REGION Network 53: Thickness AxisZ Position Absolute Position2
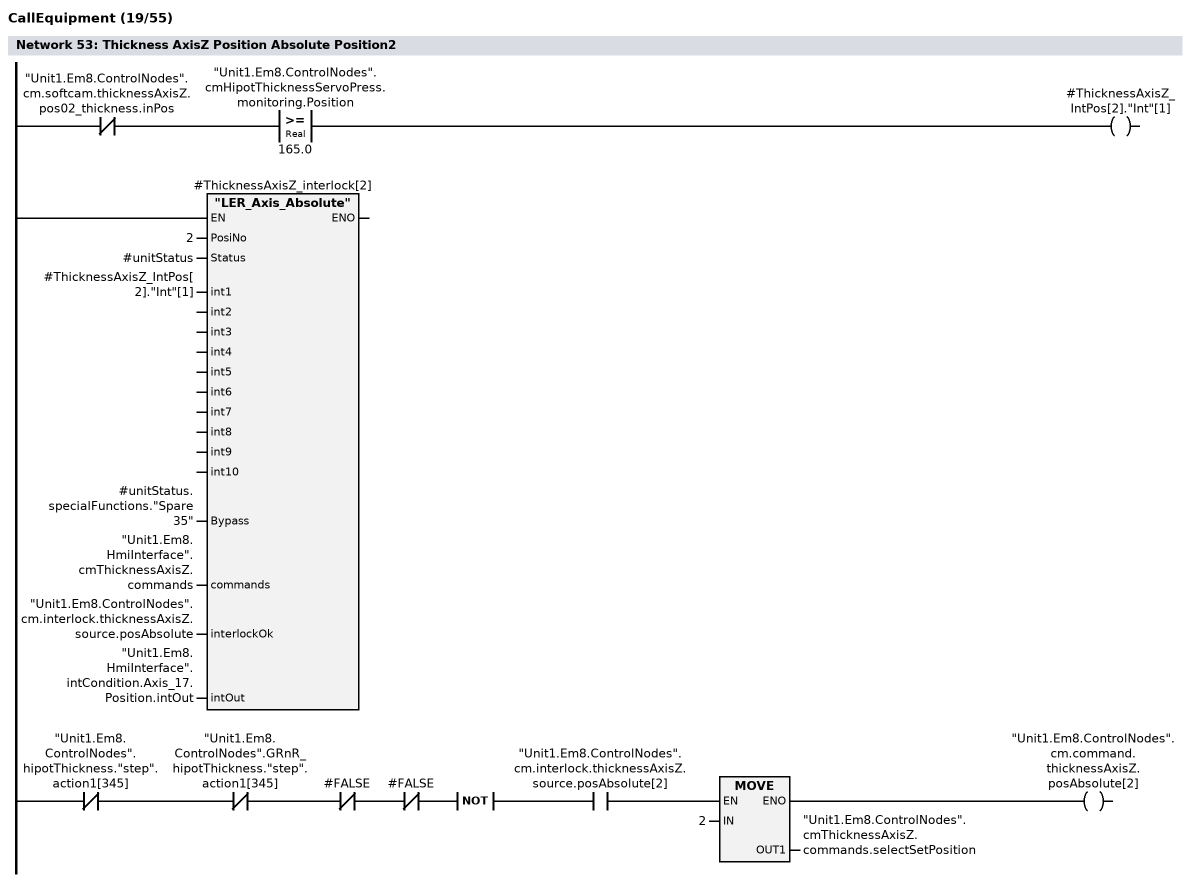
   RUNG wire#powerrail
      I_Contact( "Unit1.Em8.ControlNodes".cm.softcam.thicknessAxisZ.pos02_thickness.inPos )
      { S7_Templates := "SrcType := Real" } GE_Contact(in1 := "Unit1.Em8.ControlNodes".cmHipotThicknessServoPress.monitoring.Position, in2 := 165.0)
      Coil( #ThicknessAxisZ_IntPos[2]."Int"[1] )
   END_RUNG
   RUNG wire#powerrail
      #ThicknessAxisZ_interlock[2](PosiNo := 2, Status := #unitStatus, int1 := #ThicknessAxisZ_IntPos[2]."Int"[1], int2 :=, int3 :=, int4 :=, int5 :=, int6 :=, int7 :=, int8 :=, int9 :=, int10 :=, Bypass := #unitStatus.specialFunctions."Spare 35", commands := "Unit1.Em8.HmiInterface".cmThicknessAxisZ.commands, interlockOk := "Unit1.Em8.ControlNodes".cm.interlock.thicknessAxisZ.source.posAbsolute, intOut := "Unit1.Em8.HmiInterface".intCondition.Axis_17.Position.intOut)
   END_RUNG
   RUNG wire#powerrail
      I_Contact( "Unit1.Em8.ControlNodes".hipotThickness."step".action1[345] )
      I_Contact( "Unit1.Em8.ControlNodes".GRnR_hipotThickness."step".action1[345] )
      I_Contact( #FALSE )
      I_Contact( #FALSE )
      Not()
      Contact( "Unit1.Em8.ControlNodes".cm.interlock.thicknessAxisZ.source.posAbsolute[2] )
      Move(in := 2, out1 => "Unit1.Em8.ControlNodes".cmThicknessAxisZ.commands.selectSetPosition)
      Coil( "Unit1.Em8.ControlNodes".cm.command.thicknessAxisZ.posAbsolute[2] )
   END_RUNG
   // the same network as SCL:
   #ThicknessAxisZ_IntPos[2]."Int"[1] := NOT "Unit1.Em8.ControlNodes".cm.softcam.thicknessAxisZ.pos02_thickness.inPos AND ("Unit1.Em8.ControlNodes".cmHipotThicknessServoPress.monitoring.Position >= 165.0);
   #ThicknessAxisZ_interlock[2](PosiNo := 2,   // "LER_Axis_Absolute"
                           Status := #unitStatus,
                           int1 := #ThicknessAxisZ_IntPos[2]."Int"[1],
                           Bypass := #unitStatus.specialFunctions."Spare 35",
                           commands := "Unit1.Em8.HmiInterface".cmThicknessAxisZ.commands,
                           interlockOk := "Unit1.Em8.ControlNodes".cm.interlock.thicknessAxisZ.source.posAbsolute,
                           intOut := "Unit1.Em8.HmiInterface".intCondition.Axis_17.Position.intOut);
   #_w1 := NOT (NOT "Unit1.Em8.ControlNodes".hipotThickness."step".action1[345] AND NOT "Unit1.Em8.ControlNodes".GRnR_hipotThickness."step".action1[345] AND NOT #FALSE AND NOT #FALSE) AND "Unit1.Em8.ControlNodes".cm.interlock.thicknessAxisZ.source.posAbsolute[2];
   IF #_w1 THEN "Unit1.Em8.ControlNodes".cmThicknessAxisZ.commands.selectSetPosition := 2; END_IF;
   "Unit1.Em8.ControlNodes".cm.command.thicknessAxisZ.posAbsolute[2] := #_w1;
END_REGION

REGION Network 54: Thickness AxisZ Position Absolute Position3
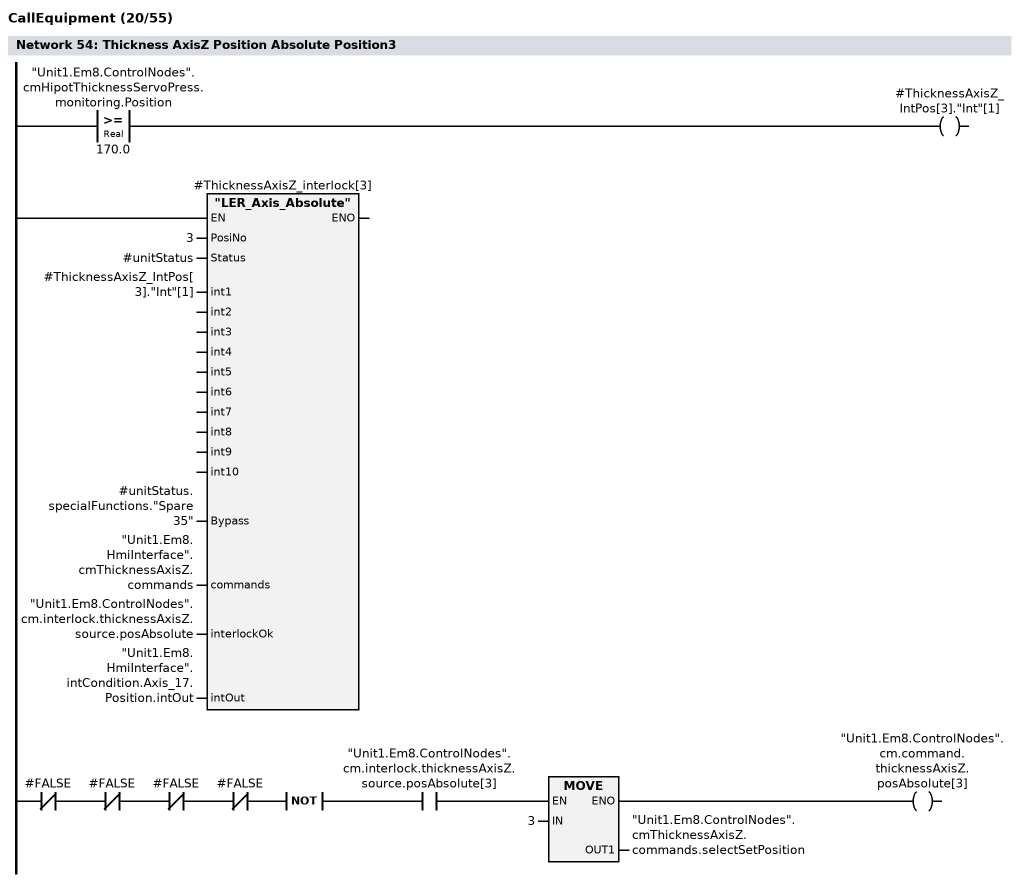
   RUNG wire#powerrail
      { S7_Templates := "SrcType := Real" } GE_Contact(in1 := "Unit1.Em8.ControlNodes".cmHipotThicknessServoPress.monitoring.Position, in2 := 170.0)
      Coil( #ThicknessAxisZ_IntPos[3]."Int"[1] )
   END_RUNG
   RUNG wire#powerrail
      #ThicknessAxisZ_interlock[3](PosiNo := 3, Status := #unitStatus, int1 := #ThicknessAxisZ_IntPos[3]."Int"[1], int2 :=, int3 :=, int4 :=, int5 :=, int6 :=, int7 :=, int8 :=, int9 :=, int10 :=, Bypass := #unitStatus.specialFunctions."Spare 35", commands := "Unit1.Em8.HmiInterface".cmThicknessAxisZ.commands, interlockOk := "Unit1.Em8.ControlNodes".cm.interlock.thicknessAxisZ.source.posAbsolute, intOut := "Unit1.Em8.HmiInterface".intCondition.Axis_17.Position.intOut)
   END_RUNG
   RUNG wire#powerrail
      I_Contact( #FALSE )
      I_Contact( #FALSE )
      I_Contact( #FALSE )
      I_Contact( #FALSE )
      Not()
      Contact( "Unit1.Em8.ControlNodes".cm.interlock.thicknessAxisZ.source.posAbsolute[3] )
      Move(in := 3, out1 => "Unit1.Em8.ControlNodes".cmThicknessAxisZ.commands.selectSetPosition)
      Coil( "Unit1.Em8.ControlNodes".cm.command.thicknessAxisZ.posAbsolute[3] )
   END_RUNG
   // the same network as SCL:
   #ThicknessAxisZ_IntPos[3]."Int"[1] := "Unit1.Em8.ControlNodes".cmHipotThicknessServoPress.monitoring.Position >= 170.0;
   #ThicknessAxisZ_interlock[3](PosiNo := 3,   // "LER_Axis_Absolute"
                           Status := #unitStatus,
                           int1 := #ThicknessAxisZ_IntPos[3]."Int"[1],
                           Bypass := #unitStatus.specialFunctions."Spare 35",
                           commands := "Unit1.Em8.HmiInterface".cmThicknessAxisZ.commands,
                           interlockOk := "Unit1.Em8.ControlNodes".cm.interlock.thicknessAxisZ.source.posAbsolute,
                           intOut := "Unit1.Em8.HmiInterface".intCondition.Axis_17.Position.intOut);
   #_w1 := NOT (NOT #FALSE AND NOT #FALSE AND NOT #FALSE AND NOT #FALSE) AND "Unit1.Em8.ControlNodes".cm.interlock.thicknessAxisZ.source.posAbsolute[3];
   IF #_w1 THEN "Unit1.Em8.ControlNodes".cmThicknessAxisZ.commands.selectSetPosition := 3; END_IF;
   "Unit1.Em8.ControlNodes".cm.command.thicknessAxisZ.posAbsolute[3] := #_w1;
END_REGION

REGION Network 55: Thickness AxisZ Position Absolute Position4
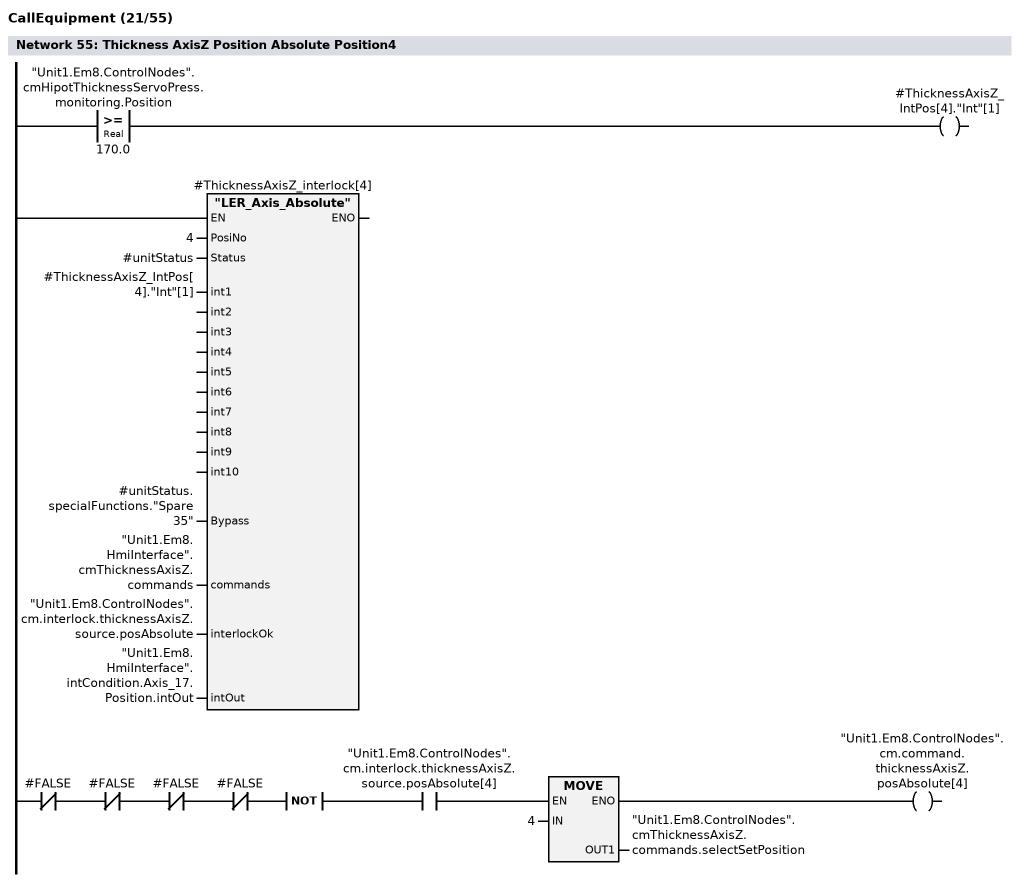
   RUNG wire#powerrail
      { S7_Templates := "SrcType := Real" } GE_Contact(in1 := "Unit1.Em8.ControlNodes".cmHipotThicknessServoPress.monitoring.Position, in2 := 170.0)
      Coil( #ThicknessAxisZ_IntPos[4]."Int"[1] )
   END_RUNG
   RUNG wire#powerrail
      #ThicknessAxisZ_interlock[4](PosiNo := 4, Status := #unitStatus, int1 := #ThicknessAxisZ_IntPos[4]."Int"[1], int2 :=, int3 :=, int4 :=, int5 :=, int6 :=, int7 :=, int8 :=, int9 :=, int10 :=, Bypass := #unitStatus.specialFunctions."Spare 35", commands := "Unit1.Em8.HmiInterface".cmThicknessAxisZ.commands, interlockOk := "Unit1.Em8.ControlNodes".cm.interlock.thicknessAxisZ.source.posAbsolute, intOut := "Unit1.Em8.HmiInterface".intCondition.Axis_17.Position.intOut)
   END_RUNG
   RUNG wire#powerrail
      I_Contact( #FALSE )
      I_Contact( #FALSE )
      I_Contact( #FALSE )
      I_Contact( #FALSE )
      Not()
      Contact( "Unit1.Em8.ControlNodes".cm.interlock.thicknessAxisZ.source.posAbsolute[4] )
      Move(in := 4, out1 => "Unit1.Em8.ControlNodes".cmThicknessAxisZ.commands.selectSetPosition)
      Coil( "Unit1.Em8.ControlNodes".cm.command.thicknessAxisZ.posAbsolute[4] )
   END_RUNG
   // the same network as SCL:
   #ThicknessAxisZ_IntPos[4]."Int"[1] := "Unit1.Em8.ControlNodes".cmHipotThicknessServoPress.monitoring.Position >= 170.0;
   #ThicknessAxisZ_interlock[4](PosiNo := 4,   // "LER_Axis_Absolute"
                           Status := #unitStatus,
                           int1 := #ThicknessAxisZ_IntPos[4]."Int"[1],
                           Bypass := #unitStatus.specialFunctions."Spare 35",
                           commands := "Unit1.Em8.HmiInterface".cmThicknessAxisZ.commands,
                           interlockOk := "Unit1.Em8.ControlNodes".cm.interlock.thicknessAxisZ.source.posAbsolute,
                           intOut := "Unit1.Em8.HmiInterface".intCondition.Axis_17.Position.intOut);
   #_w1 := NOT (NOT #FALSE AND NOT #FALSE AND NOT #FALSE AND NOT #FALSE) AND "Unit1.Em8.ControlNodes".cm.interlock.thicknessAxisZ.source.posAbsolute[4];
   IF #_w1 THEN "Unit1.Em8.ControlNodes".cmThicknessAxisZ.commands.selectSetPosition := 4; END_IF;
   "Unit1.Em8.ControlNodes".cm.command.thicknessAxisZ.posAbsolute[4] := #_w1;
END_REGION

REGION Network 56: Thickness AxisZ Position Absolute Position5
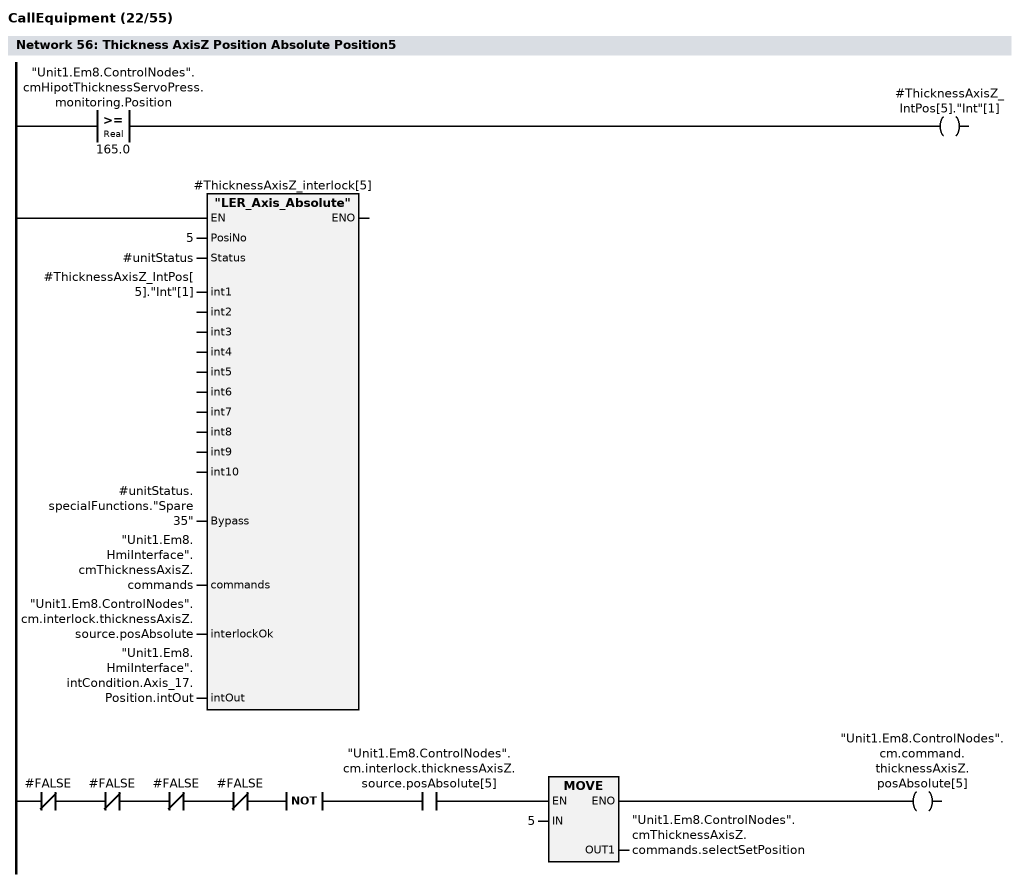
   RUNG wire#powerrail
      { S7_Templates := "SrcType := Real" } GE_Contact(in1 := "Unit1.Em8.ControlNodes".cmHipotThicknessServoPress.monitoring.Position, in2 := 165.0)
      Coil( #ThicknessAxisZ_IntPos[5]."Int"[1] )
   END_RUNG
   RUNG wire#powerrail
      #ThicknessAxisZ_interlock[5](PosiNo := 5, Status := #unitStatus, int1 := #ThicknessAxisZ_IntPos[5]."Int"[1], int2 :=, int3 :=, int4 :=, int5 :=, int6 :=, int7 :=, int8 :=, int9 :=, int10 :=, Bypass := #unitStatus.specialFunctions."Spare 35", commands := "Unit1.Em8.HmiInterface".cmThicknessAxisZ.commands, interlockOk := "Unit1.Em8.ControlNodes".cm.interlock.thicknessAxisZ.source.posAbsolute, intOut := "Unit1.Em8.HmiInterface".intCondition.Axis_17.Position.intOut)
   END_RUNG
   RUNG wire#powerrail
      I_Contact( #FALSE )
      I_Contact( #FALSE )
      I_Contact( #FALSE )
      I_Contact( #FALSE )
      Not()
      Contact( "Unit1.Em8.ControlNodes".cm.interlock.thicknessAxisZ.source.posAbsolute[5] )
      Move(in := 5, out1 => "Unit1.Em8.ControlNodes".cmThicknessAxisZ.commands.selectSetPosition)
      Coil( "Unit1.Em8.ControlNodes".cm.command.thicknessAxisZ.posAbsolute[5] )
   END_RUNG
   // the same network as SCL:
   #ThicknessAxisZ_IntPos[5]."Int"[1] := "Unit1.Em8.ControlNodes".cmHipotThicknessServoPress.monitoring.Position >= 165.0;
   #ThicknessAxisZ_interlock[5](PosiNo := 5,   // "LER_Axis_Absolute"
                           Status := #unitStatus,
                           int1 := #ThicknessAxisZ_IntPos[5]."Int"[1],
                           Bypass := #unitStatus.specialFunctions."Spare 35",
                           commands := "Unit1.Em8.HmiInterface".cmThicknessAxisZ.commands,
                           interlockOk := "Unit1.Em8.ControlNodes".cm.interlock.thicknessAxisZ.source.posAbsolute,
                           intOut := "Unit1.Em8.HmiInterface".intCondition.Axis_17.Position.intOut);
   #_w1 := NOT (NOT #FALSE AND NOT #FALSE AND NOT #FALSE AND NOT #FALSE) AND "Unit1.Em8.ControlNodes".cm.interlock.thicknessAxisZ.source.posAbsolute[5];
   IF #_w1 THEN "Unit1.Em8.ControlNodes".cmThicknessAxisZ.commands.selectSetPosition := 5; END_IF;
   "Unit1.Em8.ControlNodes".cm.command.thicknessAxisZ.posAbsolute[5] := #_w1;
END_REGION

REGION Network 57: Thickness AxisZ Position Absolute Position7
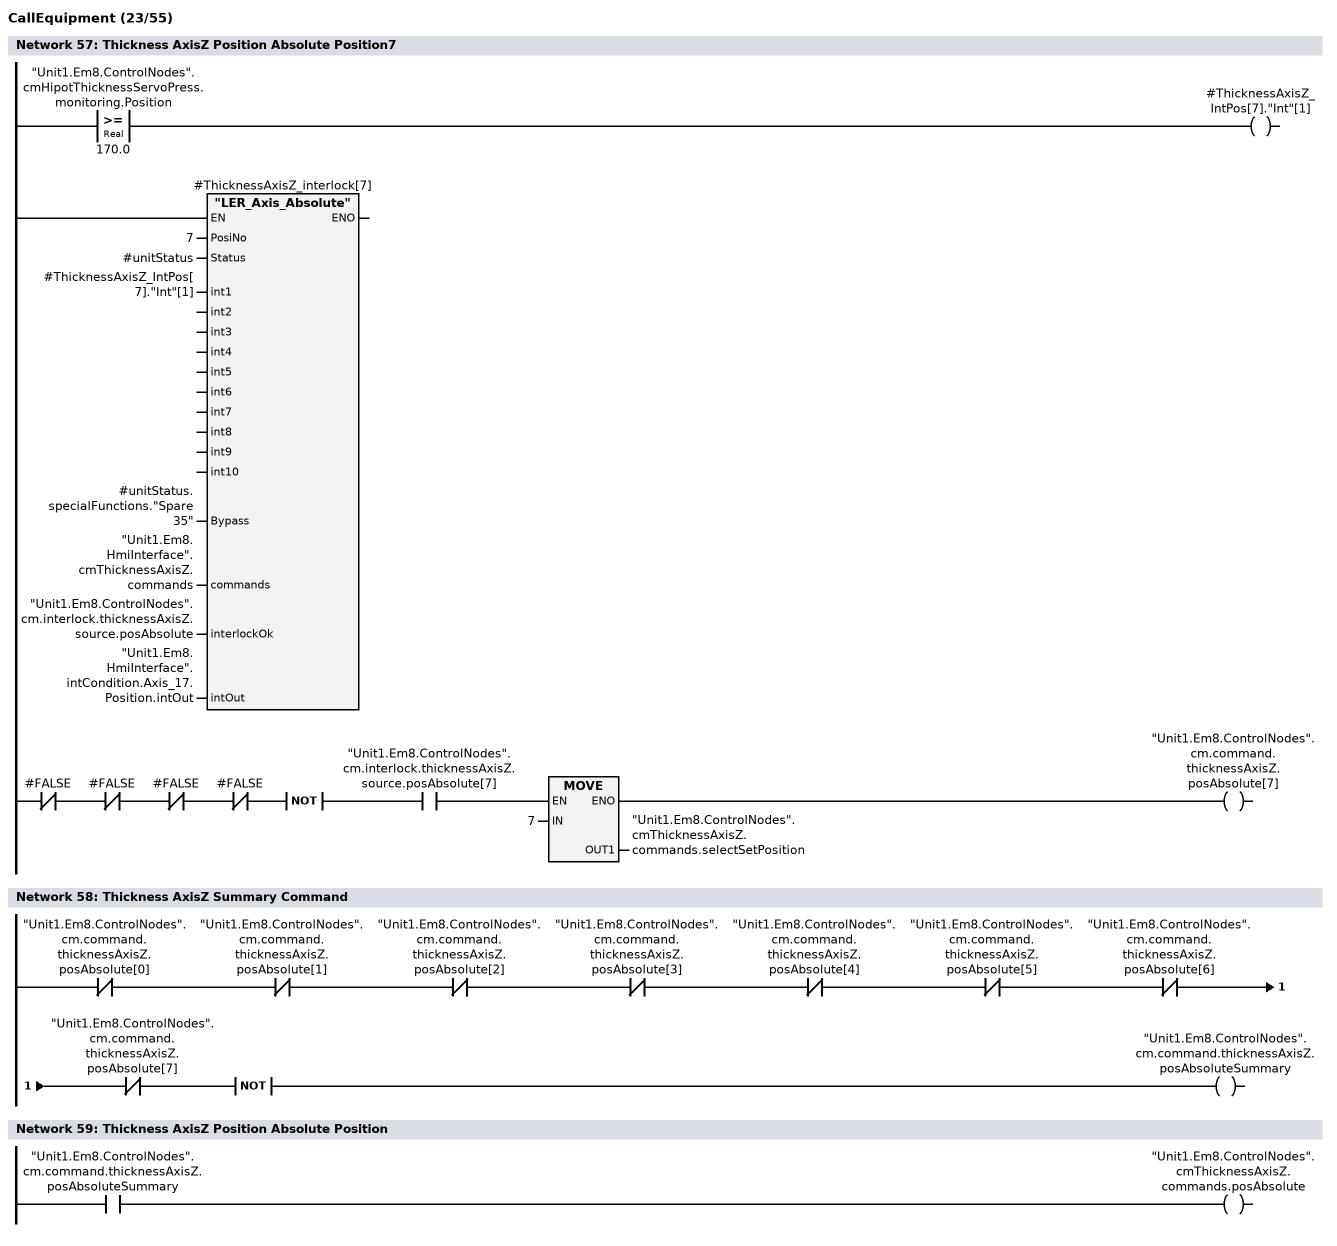
   RUNG wire#powerrail
      { S7_Templates := "SrcType := Real" } GE_Contact(in1 := "Unit1.Em8.ControlNodes".cmHipotThicknessServoPress.monitoring.Position, in2 := 170.0)
      Coil( #ThicknessAxisZ_IntPos[7]."Int"[1] )
   END_RUNG
   RUNG wire#powerrail
      #ThicknessAxisZ_interlock[7](PosiNo := 7, Status := #unitStatus, int1 := #ThicknessAxisZ_IntPos[7]."Int"[1], int2 :=, int3 :=, int4 :=, int5 :=, int6 :=, int7 :=, int8 :=, int9 :=, int10 :=, Bypass := #unitStatus.specialFunctions."Spare 35", commands := "Unit1.Em8.HmiInterface".cmThicknessAxisZ.commands, interlockOk := "Unit1.Em8.ControlNodes".cm.interlock.thicknessAxisZ.source.posAbsolute, intOut := "Unit1.Em8.HmiInterface".intCondition.Axis_17.Position.intOut)
   END_RUNG
   RUNG wire#powerrail
      I_Contact( #FALSE )
      I_Contact( #FALSE )
      I_Contact( #FALSE )
      I_Contact( #FALSE )
      Not()
      Contact( "Unit1.Em8.ControlNodes".cm.interlock.thicknessAxisZ.source.posAbsolute[7] )
      Move(in := 7, out1 => "Unit1.Em8.ControlNodes".cmThicknessAxisZ.commands.selectSetPosition)
      Coil( "Unit1.Em8.ControlNodes".cm.command.thicknessAxisZ.posAbsolute[7] )
   END_RUNG
   // the same network as SCL:
   #ThicknessAxisZ_IntPos[7]."Int"[1] := "Unit1.Em8.ControlNodes".cmHipotThicknessServoPress.monitoring.Position >= 170.0;
   #ThicknessAxisZ_interlock[7](PosiNo := 7,   // "LER_Axis_Absolute"
                           Status := #unitStatus,
                           int1 := #ThicknessAxisZ_IntPos[7]."Int"[1],
                           Bypass := #unitStatus.specialFunctions."Spare 35",
                           commands := "Unit1.Em8.HmiInterface".cmThicknessAxisZ.commands,
                           interlockOk := "Unit1.Em8.ControlNodes".cm.interlock.thicknessAxisZ.source.posAbsolute,
                           intOut := "Unit1.Em8.HmiInterface".intCondition.Axis_17.Position.intOut);
   #_w1 := NOT (NOT #FALSE AND NOT #FALSE AND NOT #FALSE AND NOT #FALSE) AND "Unit1.Em8.ControlNodes".cm.interlock.thicknessAxisZ.source.posAbsolute[7];
   IF #_w1 THEN "Unit1.Em8.ControlNodes".cmThicknessAxisZ.commands.selectSetPosition := 7; END_IF;
   "Unit1.Em8.ControlNodes".cm.command.thicknessAxisZ.posAbsolute[7] := #_w1;
END_REGION

REGION Network 58: Thickness AxisZ Summary Command
   RUNG wire#powerrail
      I_Contact( "Unit1.Em8.ControlNodes".cm.command.thicknessAxisZ.posAbsolute[0] )
      I_Contact( "Unit1.Em8.ControlNodes".cm.command.thicknessAxisZ.posAbsolute[1] )
      I_Contact( "Unit1.Em8.ControlNodes".cm.command.thicknessAxisZ.posAbsolute[2] )
      I_Contact( "Unit1.Em8.ControlNodes".cm.command.thicknessAxisZ.posAbsolute[3] )
      I_Contact( "Unit1.Em8.ControlNodes".cm.command.thicknessAxisZ.posAbsolute[4] )
      I_Contact( "Unit1.Em8.ControlNodes".cm.command.thicknessAxisZ.posAbsolute[5] )
      I_Contact( "Unit1.Em8.ControlNodes".cm.command.thicknessAxisZ.posAbsolute[6] )
      I_Contact( "Unit1.Em8.ControlNodes".cm.command.thicknessAxisZ.posAbsolute[7] )
      Not()
      Coil( "Unit1.Em8.ControlNodes".cm.command.thicknessAxisZ.posAbsoluteSummary )
   END_RUNG
   // the same network as SCL:
   "Unit1.Em8.ControlNodes".cm.command.thicknessAxisZ.posAbsoluteSummary := NOT (NOT "Unit1.Em8.ControlNodes".cm.command.thicknessAxisZ.posAbsolute[0] AND NOT "Unit1.Em8.ControlNodes".cm.command.thicknessAxisZ.posAbsolute[1] AND NOT "Unit1.Em8.ControlNodes".cm.command.thicknessAxisZ.posAbsolute[2] AND NOT "Unit1.Em8.ControlNodes".cm.command.thicknessAxisZ.posAbsolute[3] AND NOT "Unit1.Em8.ControlNodes".cm.command.thicknessAxisZ.posAbsolute[4] AND NOT "Unit1.Em8.ControlNodes".cm.command.thicknessAxisZ.posAbsolute[5] AND NOT "Unit1.Em8.ControlNodes".cm.command.thicknessAxisZ.posAbsolute[6] AND NOT "Unit1.Em8.ControlNodes".cm.command.thicknessAxisZ.posAbsolute[7]);
END_REGION

REGION Network 59: Thickness AxisZ Position Absolute Position
   RUNG wire#powerrail
      Contact( "Unit1.Em8.ControlNodes".cm.command.thicknessAxisZ.posAbsoluteSummary )
      Coil( "Unit1.Em8.ControlNodes".cmThicknessAxisZ.commands.posAbsolute )
   END_RUNG
   // the same network as SCL:
   "Unit1.Em8.ControlNodes".cmThicknessAxisZ.commands.posAbsolute := "Unit1.Em8.ControlNodes".cm.command.thicknessAxisZ.posAbsoluteSummary;
END_REGION

REGION Network 60: Thickness AxisZ Interlock Summary
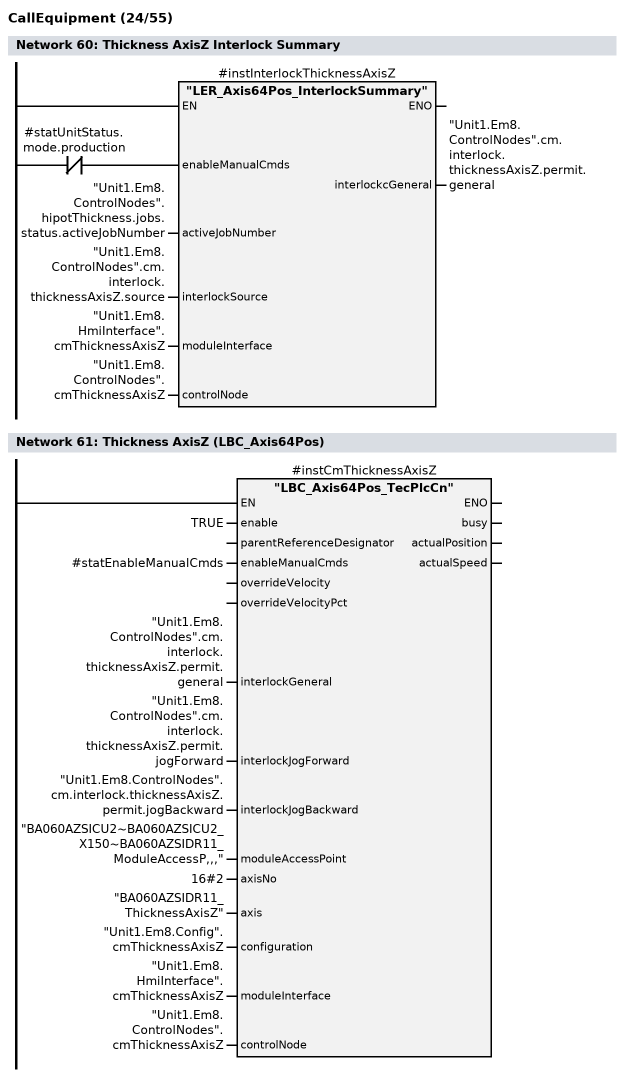
   RUNG wire#powerrail
      #instInterlockThicknessAxisZ(enableManualCmds := wire#w1, activeJobNumber := "Unit1.Em8.ControlNodes".hipotThickness.jobs.status.activeJobNumber, interlockSource := "Unit1.Em8.ControlNodes".cm.interlock.thicknessAxisZ.source, moduleInterface := "Unit1.Em8.HmiInterface".cmThicknessAxisZ, controlNode := "Unit1.Em8.ControlNodes".cmThicknessAxisZ, interlockcGeneral => "Unit1.Em8.ControlNodes".cm.interlock.thicknessAxisZ.permit.general)
   END_RUNG
   RUNG wire#powerrail
      I_Contact( #statUnitStatus.mode.production )
   END_RUNG wire#w1
   // the same network as SCL:
   #instInterlockThicknessAxisZ(enableManualCmds := NOT #statUnitStatus.mode.production,   // "LER_Axis64Pos_InterlockSummary"
                           activeJobNumber := "Unit1.Em8.ControlNodes".hipotThickness.jobs.status.activeJobNumber,
                           interlockSource := "Unit1.Em8.ControlNodes".cm.interlock.thicknessAxisZ.source,
                           moduleInterface := "Unit1.Em8.HmiInterface".cmThicknessAxisZ,
                           controlNode := "Unit1.Em8.ControlNodes".cmThicknessAxisZ,
                           interlockcGeneral => "Unit1.Em8.ControlNodes".cm.interlock.thicknessAxisZ.permit.general);
END_REGION

REGION Network 61: Thickness AxisZ (LBC_Axis64Pos)
   RUNG wire#powerrail
      #instCmThicknessAxisZ(enable := TRUE, parentReferenceDesignator :=, enableManualCmds := #statEnableManualCmds, overrideVelocity :=, overrideVelocityPct :=, interlockGeneral := "Unit1.Em8.ControlNodes".cm.interlock.thicknessAxisZ.permit.general, interlockJogForward := "Unit1.Em8.ControlNodes".cm.interlock.thicknessAxisZ.permit.jogForward, interlockJogBackward := "Unit1.Em8.ControlNodes".cm.interlock.thicknessAxisZ.permit.jogBackward, moduleAccessPoint := "BA060AZSICU2~BA060AZSICU2_X150~BA060AZSIDR11_ModuleAccessP,,,", axisNo := 16#2, axis := "BA060AZSIDR11_ThicknessAxisZ", configuration := "Unit1.Em8.Config".cmThicknessAxisZ, moduleInterface := "Unit1.Em8.HmiInterface".cmThicknessAxisZ, controlNode := "Unit1.Em8.ControlNodes".cmThicknessAxisZ, busy =>, actualPosition =>, actualSpeed =>)
   END_RUNG
   // the same network as SCL:
   #instCmThicknessAxisZ(enable := TRUE,   // "LBC_Axis64Pos_TecPlcCn"
                         enableManualCmds := #statEnableManualCmds,
                         interlockGeneral := "Unit1.Em8.ControlNodes".cm.interlock.thicknessAxisZ.permit.general,
                         interlockJogForward := "Unit1.Em8.ControlNodes".cm.interlock.thicknessAxisZ.permit.jogForward,
                         interlockJogBackward := "Unit1.Em8.ControlNodes".cm.interlock.thicknessAxisZ.permit.jogBackward,
                         moduleAccessPoint := "BA060AZSICU2~BA060AZSICU2_X150~BA060AZSIDR11_ModuleAccessP,,,",
                         axisNo := 16#2,
                         axis := "BA060AZSIDR11_ThicknessAxisZ",
                         configuration := "Unit1.Em8.Config".cmThicknessAxisZ,
                         moduleInterface := "Unit1.Em8.HmiInterface".cmThicknessAxisZ,
                         controlNode := "Unit1.Em8.ControlNodes".cmThicknessAxisZ);
END_REGION

REGION Network 62: Thickness AxisZ Softcam
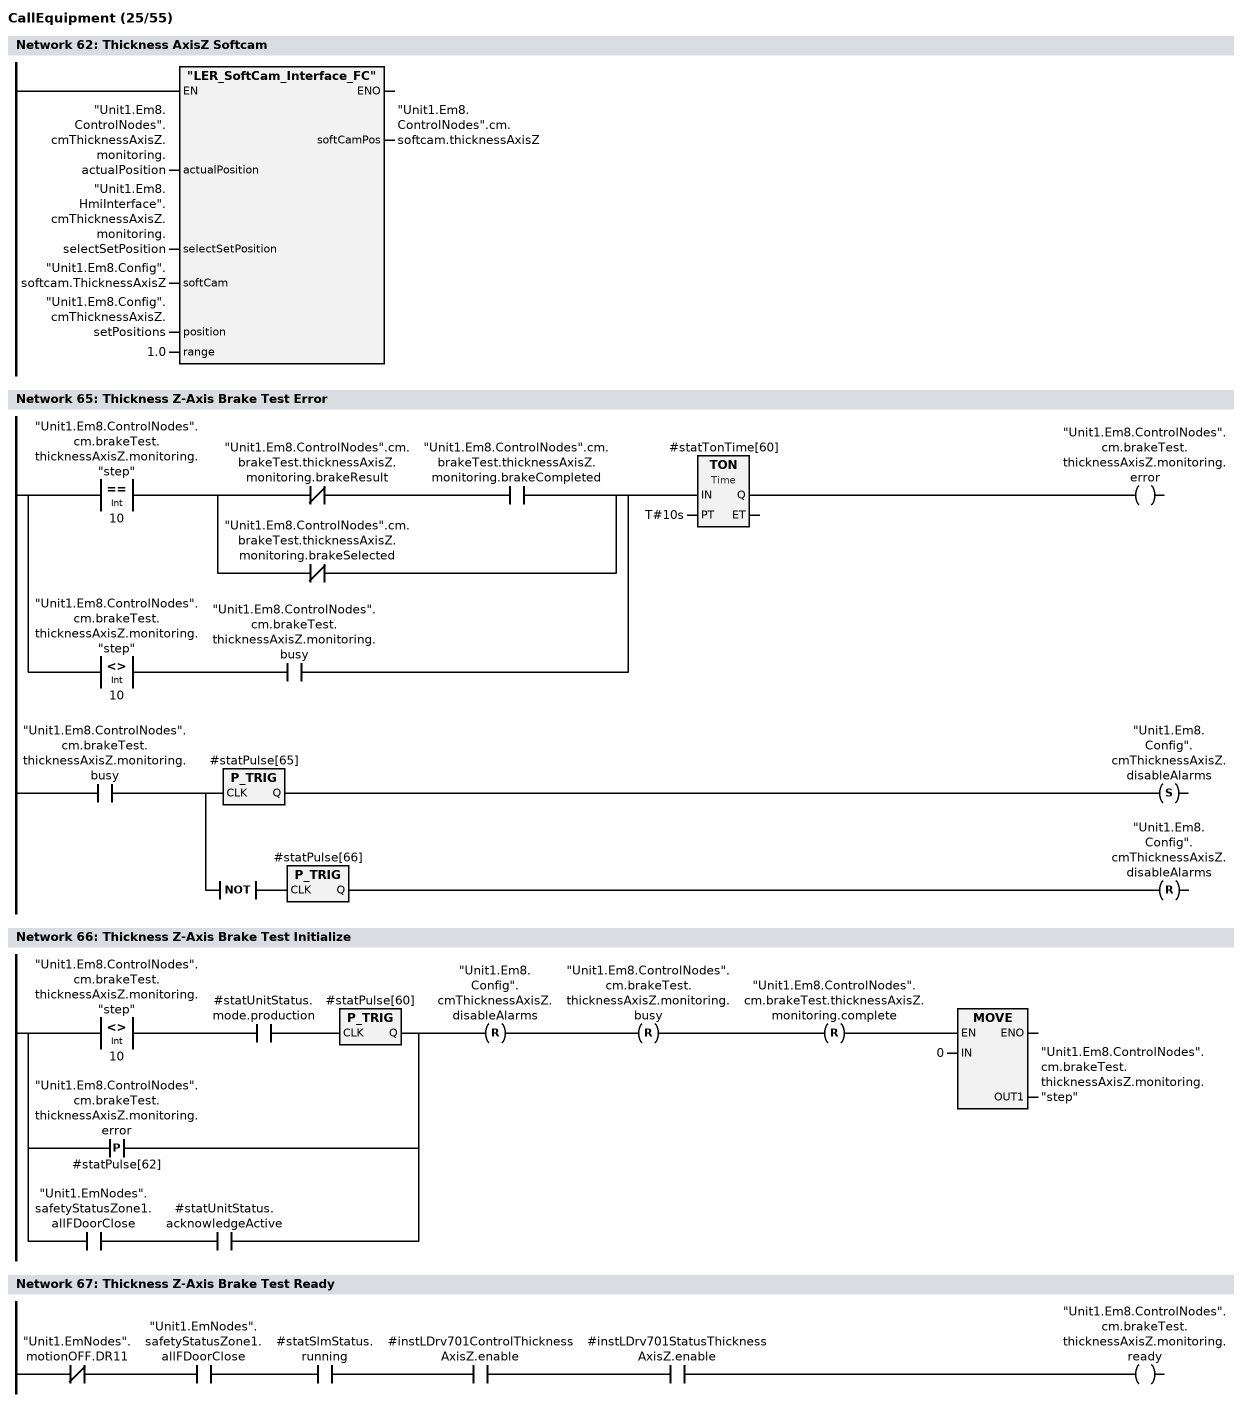
   RUNG wire#powerrail
      "LER_SoftCam_Interface_FC"(actualPosition := "Unit1.Em8.ControlNodes".cmThicknessAxisZ.monitoring.actualPosition, selectSetPosition := "Unit1.Em8.HmiInterface".cmThicknessAxisZ.monitoring.selectSetPosition, softCam := "Unit1.Em8.Config".softcam.ThicknessAxisZ, position := "Unit1.Em8.Config".cmThicknessAxisZ.setPositions, range := 1.0, softCamPos => "Unit1.Em8.ControlNodes".cm.softcam.thicknessAxisZ)
   END_RUNG
   // the same network as SCL:
   "LER_SoftCam_Interface_FC"(actualPosition := "Unit1.Em8.ControlNodes".cmThicknessAxisZ.monitoring.actualPosition,
                           selectSetPosition := "Unit1.Em8.HmiInterface".cmThicknessAxisZ.monitoring.selectSetPosition,
                           softCam := "Unit1.Em8.Config".softcam.ThicknessAxisZ,
                           position := "Unit1.Em8.Config".cmThicknessAxisZ.setPositions,
                           range := 1.0,
                           softCamPos => "Unit1.Em8.ControlNodes".cm.softcam.thicknessAxisZ);
END_REGION

REGION Network 64: ******************** Brake Test (Axis) ********************
END_REGION

REGION Network 65: Thickness Z-Axis Brake Test Error
   RUNG wire#powerrail
      { S7_Templates := "SrcType := Int" } EQ_Contact(in1 := "Unit1.Em8.ControlNodes".cm.brakeTest.thicknessAxisZ.monitoring."step", in2 := 10)
      wire#w1
      I_Contact( "Unit1.Em8.ControlNodes".cm.brakeTest.thicknessAxisZ.monitoring.brakeResult )
      Contact( "Unit1.Em8.ControlNodes".cm.brakeTest.thicknessAxisZ.monitoring.brakeCompleted )
      wire#w2
      { S7_Templates := "time_type := Time" } #statTonTime[60].TON(pt := T#10s, et =>)
      Coil( "Unit1.Em8.ControlNodes".cm.brakeTest.thicknessAxisZ.monitoring.error )
   END_RUNG
   RUNG wire#w1
      I_Contact( "Unit1.Em8.ControlNodes".cm.brakeTest.thicknessAxisZ.monitoring.brakeSelected )
   END_RUNG wire#w2
   RUNG wire#powerrail
      { S7_Templates := "SrcType := Int" } NE_Contact(in1 := "Unit1.Em8.ControlNodes".cm.brakeTest.thicknessAxisZ.monitoring."step", in2 := 10)
      Contact( "Unit1.Em8.ControlNodes".cm.brakeTest.thicknessAxisZ.monitoring.busy )
   END_RUNG wire#w2
   RUNG wire#powerrail
      Contact( "Unit1.Em8.ControlNodes".cm.brakeTest.thicknessAxisZ.monitoring.busy )
      wire#w3
      P_Trig( #statPulse[65] )
      S_Coil( "Unit1.Em8.Config".cmThicknessAxisZ.disableAlarms )
   END_RUNG
   RUNG wire#w3
      Not()
      P_Trig( #statPulse[66] )
      R_Coil( "Unit1.Em8.Config".cmThicknessAxisZ.disableAlarms )
   END_RUNG
   // the same network as SCL:
   #statTonTime[60].TON(IN := (("Unit1.Em8.ControlNodes".cm.brakeTest.thicknessAxisZ.monitoring."step" = 10) AND ((NOT "Unit1.Em8.ControlNodes".cm.brakeTest.thicknessAxisZ.monitoring.brakeResult AND "Unit1.Em8.ControlNodes".cm.brakeTest.thicknessAxisZ.monitoring.brakeCompleted) OR NOT "Unit1.Em8.ControlNodes".cm.brakeTest.thicknessAxisZ.monitoring.brakeSelected)) OR (("Unit1.Em8.ControlNodes".cm.brakeTest.thicknessAxisZ.monitoring."step" <> 10) AND "Unit1.Em8.ControlNodes".cm.brakeTest.thicknessAxisZ.monitoring.busy),
                        PT := T#10s);
   "Unit1.Em8.ControlNodes".cm.brakeTest.thicknessAxisZ.monitoring.error := #statTonTime[60].Q;
   #_w1 := "Unit1.Em8.ControlNodes".cm.brakeTest.thicknessAxisZ.monitoring.busy AND NOT #statPulse[65];   // rising edge
   #statPulse[65] := "Unit1.Em8.ControlNodes".cm.brakeTest.thicknessAxisZ.monitoring.busy;
   IF #_w1 THEN "Unit1.Em8.Config".cmThicknessAxisZ.disableAlarms := TRUE; END_IF;
   #_w2 := NOT "Unit1.Em8.ControlNodes".cm.brakeTest.thicknessAxisZ.monitoring.busy AND NOT #statPulse[66];   // rising edge
   #statPulse[66] := NOT "Unit1.Em8.ControlNodes".cm.brakeTest.thicknessAxisZ.monitoring.busy;
   IF #_w2 THEN "Unit1.Em8.Config".cmThicknessAxisZ.disableAlarms := FALSE; END_IF;
END_REGION

REGION Network 66: Thickness Z-Axis Brake Test Initialize
   RUNG wire#powerrail
      { S7_Templates := "SrcType := Int" } NE_Contact(in1 := "Unit1.Em8.ControlNodes".cm.brakeTest.thicknessAxisZ.monitoring."step", in2 := 10)
      Contact( #statUnitStatus.mode.production )
      P_Trig( #statPulse[60] )
      wire#w1
      R_Coil( "Unit1.Em8.Config".cmThicknessAxisZ.disableAlarms )
      R_Coil( "Unit1.Em8.ControlNodes".cm.brakeTest.thicknessAxisZ.monitoring.busy )
      R_Coil( "Unit1.Em8.ControlNodes".cm.brakeTest.thicknessAxisZ.monitoring.complete )
      Move(in := 0, out1 => "Unit1.Em8.ControlNodes".cm.brakeTest.thicknessAxisZ.monitoring."step")
   END_RUNG
   RUNG wire#powerrail
      P_Contact(operand := "Unit1.Em8.ControlNodes".cm.brakeTest.thicknessAxisZ.monitoring.error, bit := #statPulse[62])
   END_RUNG wire#w1
   RUNG wire#powerrail
      Contact( "Unit1.EmNodes".safetyStatusZone1.allFDoorClose )
      Contact( #statUnitStatus.acknowledgeActive )
   END_RUNG wire#w1
   // the same network as SCL:
   #_w1 := ("Unit1.Em8.ControlNodes".cm.brakeTest.thicknessAxisZ.monitoring."step" <> 10) AND #statUnitStatus.mode.production;
   #_w2 := #_w1 AND NOT #statPulse[60];   // rising edge
   #statPulse[60] := #_w1;
   #_w3 := "Unit1.Em8.ControlNodes".cm.brakeTest.thicknessAxisZ.monitoring.error AND NOT #statPulse[62];   // rising edge of "Unit1.Em8.ControlNodes".cm.brakeTest.thicknessAxisZ.monitoring.error
   #statPulse[62] := "Unit1.Em8.ControlNodes".cm.brakeTest.thicknessAxisZ.monitoring.error;
   IF #_w2 OR #_w3 OR ("Unit1.EmNodes".safetyStatusZone1.allFDoorClose AND #statUnitStatus.acknowledgeActive) THEN
       "Unit1.Em8.Config".cmThicknessAxisZ.disableAlarms := FALSE;
       "Unit1.Em8.ControlNodes".cm.brakeTest.thicknessAxisZ.monitoring.busy := FALSE;
       "Unit1.Em8.ControlNodes".cm.brakeTest.thicknessAxisZ.monitoring.complete := FALSE;
       "Unit1.Em8.ControlNodes".cm.brakeTest.thicknessAxisZ.monitoring."step" := 0;
   END_IF;
END_REGION

REGION Network 67: Thickness Z-Axis Brake Test Ready
   RUNG wire#powerrail
      I_Contact( "Unit1.EmNodes".motionOFF.DR11 )
      Contact( "Unit1.EmNodes".safetyStatusZone1.allFDoorClose )
      Contact( #statSlmStatus.running )
      Contact( #instLDrv701ControlThicknessAxisZ.enable )
      Contact( #instLDrv701StatusThicknessAxisZ.enable )
      Coil( "Unit1.Em8.ControlNodes".cm.brakeTest.thicknessAxisZ.monitoring.ready )
   END_RUNG
   // the same network as SCL:
   "Unit1.Em8.ControlNodes".cm.brakeTest.thicknessAxisZ.monitoring.ready := NOT "Unit1.EmNodes".motionOFF.DR11 AND "Unit1.EmNodes".safetyStatusZone1.allFDoorClose AND #statSlmStatus.running AND #instLDrv701ControlThicknessAxisZ.enable AND #instLDrv701StatusThicknessAxisZ.enable;
END_REGION

REGION Network 68: Thickness Z-Axis Brake Test Commands
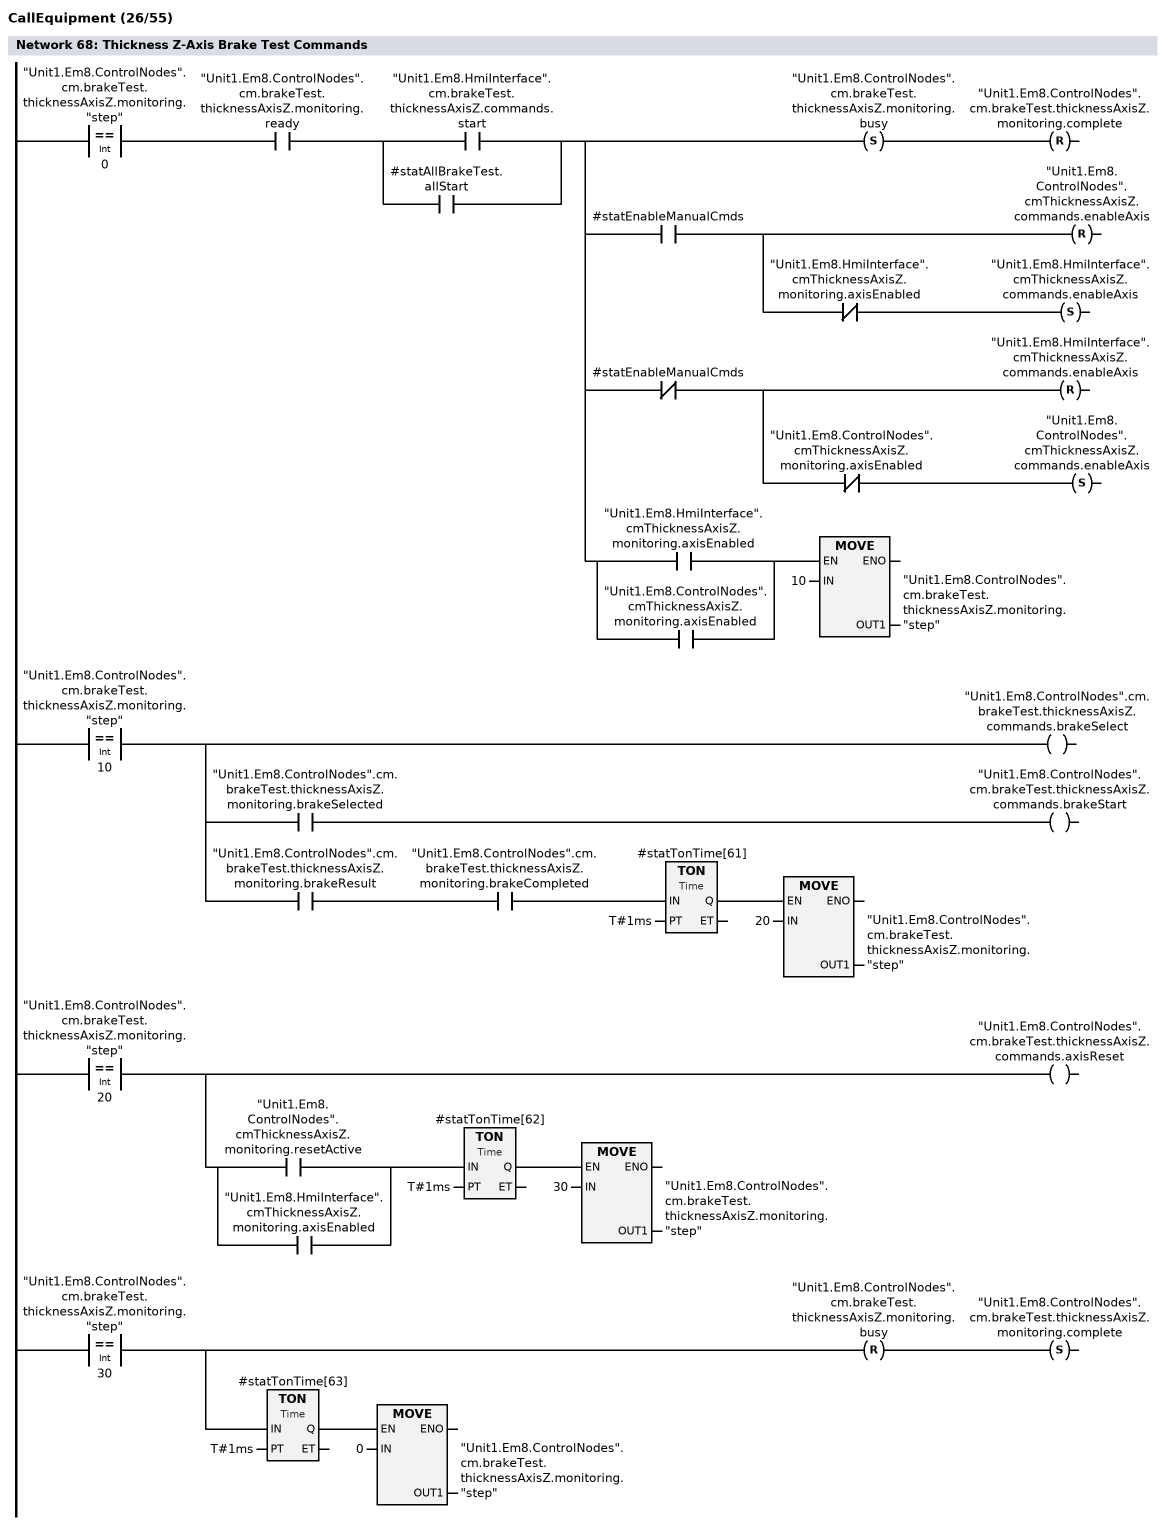
   RUNG wire#powerrail
      { S7_Templates := "SrcType := Int" } EQ_Contact(in1 := "Unit1.Em8.ControlNodes".cm.brakeTest.thicknessAxisZ.monitoring."step", in2 := 0)
      Contact( "Unit1.Em8.ControlNodes".cm.brakeTest.thicknessAxisZ.monitoring.ready )
      wire#w1
      Contact( "Unit1.Em8.HmiInterface".cm.brakeTest.thicknessAxisZ.commands.start )
      wire#w2
      S_Coil( "Unit1.Em8.ControlNodes".cm.brakeTest.thicknessAxisZ.monitoring.busy )
      R_Coil( "Unit1.Em8.ControlNodes".cm.brakeTest.thicknessAxisZ.monitoring.complete )
   END_RUNG
   RUNG wire#w1
      Contact( #statAllBrakeTest.allStart )
   END_RUNG wire#w2
   RUNG wire#w2
      Contact( #statEnableManualCmds )
      wire#w3
      R_Coil( "Unit1.Em8.ControlNodes".cmThicknessAxisZ.commands.enableAxis )
   END_RUNG
   RUNG wire#w3
      I_Contact( "Unit1.Em8.HmiInterface".cmThicknessAxisZ.monitoring.axisEnabled )
      S_Coil( "Unit1.Em8.HmiInterface".cmThicknessAxisZ.commands.enableAxis )
   END_RUNG
   RUNG wire#w2
      I_Contact( #statEnableManualCmds )
      wire#w4
      R_Coil( "Unit1.Em8.HmiInterface".cmThicknessAxisZ.commands.enableAxis )
   END_RUNG
   RUNG wire#w4
      I_Contact( "Unit1.Em8.ControlNodes".cmThicknessAxisZ.monitoring.axisEnabled )
      S_Coil( "Unit1.Em8.ControlNodes".cmThicknessAxisZ.commands.enableAxis )
   END_RUNG
   RUNG wire#w2
      Contact( "Unit1.Em8.HmiInterface".cmThicknessAxisZ.monitoring.axisEnabled )
      wire#w5
      Move(in := 10, out1 => "Unit1.Em8.ControlNodes".cm.brakeTest.thicknessAxisZ.monitoring."step")
   END_RUNG
   RUNG wire#w2
      Contact( "Unit1.Em8.ControlNodes".cmThicknessAxisZ.monitoring.axisEnabled )
   END_RUNG wire#w5
   RUNG wire#powerrail
      { S7_Templates := "SrcType := Int" } EQ_Contact(in1 := "Unit1.Em8.ControlNodes".cm.brakeTest.thicknessAxisZ.monitoring."step", in2 := 10)
      wire#w6
      Coil( "Unit1.Em8.ControlNodes".cm.brakeTest.thicknessAxisZ.commands.brakeSelect )
   END_RUNG
   RUNG wire#w6
      Contact( "Unit1.Em8.ControlNodes".cm.brakeTest.thicknessAxisZ.monitoring.brakeSelected )
      Coil( "Unit1.Em8.ControlNodes".cm.brakeTest.thicknessAxisZ.commands.brakeStart )
   END_RUNG
   RUNG wire#w6
      Contact( "Unit1.Em8.ControlNodes".cm.brakeTest.thicknessAxisZ.monitoring.brakeResult )
      Contact( "Unit1.Em8.ControlNodes".cm.brakeTest.thicknessAxisZ.monitoring.brakeCompleted )
      { S7_Templates := "time_type := Time" } #statTonTime[61].TON(pt := T#1ms, et =>)
      Move(in := 20, out1 => "Unit1.Em8.ControlNodes".cm.brakeTest.thicknessAxisZ.monitoring."step")
   END_RUNG
   RUNG wire#powerrail
      { S7_Templates := "SrcType := Int" } EQ_Contact(in1 := "Unit1.Em8.ControlNodes".cm.brakeTest.thicknessAxisZ.monitoring."step", in2 := 20)
      wire#w7
      Coil( "Unit1.Em8.ControlNodes".cm.brakeTest.thicknessAxisZ.commands.axisReset )
   END_RUNG
   RUNG wire#w7
      Contact( "Unit1.Em8.ControlNodes".cmThicknessAxisZ.monitoring.resetActive )
      wire#w8
      { S7_Templates := "time_type := Time" } #statTonTime[62].TON(pt := T#1ms, et =>)
      Move(in := 30, out1 => "Unit1.Em8.ControlNodes".cm.brakeTest.thicknessAxisZ.monitoring."step")
   END_RUNG
   RUNG wire#w7
      Contact( "Unit1.Em8.HmiInterface".cmThicknessAxisZ.monitoring.axisEnabled )
   END_RUNG wire#w8
   RUNG wire#powerrail
      { S7_Templates := "SrcType := Int" } EQ_Contact(in1 := "Unit1.Em8.ControlNodes".cm.brakeTest.thicknessAxisZ.monitoring."step", in2 := 30)
      wire#w9
      R_Coil( "Unit1.Em8.ControlNodes".cm.brakeTest.thicknessAxisZ.monitoring.busy )
      S_Coil( "Unit1.Em8.ControlNodes".cm.brakeTest.thicknessAxisZ.monitoring.complete )
   END_RUNG
   RUNG wire#w9
      { S7_Templates := "time_type := Time" } #statTonTime[63].TON(pt := T#1ms, et =>)
      Move(in := 0, out1 => "Unit1.Em8.ControlNodes".cm.brakeTest.thicknessAxisZ.monitoring."step")
   END_RUNG
   // the same network as SCL:
   #_w1 := ("Unit1.Em8.ControlNodes".cm.brakeTest.thicknessAxisZ.monitoring."step" = 0) AND "Unit1.Em8.ControlNodes".cm.brakeTest.thicknessAxisZ.monitoring.ready AND ("Unit1.Em8.HmiInterface".cm.brakeTest.thicknessAxisZ.commands.start OR #statAllBrakeTest.allStart);
   IF #_w1 THEN
       "Unit1.Em8.ControlNodes".cm.brakeTest.thicknessAxisZ.monitoring.busy := TRUE;
       "Unit1.Em8.ControlNodes".cm.brakeTest.thicknessAxisZ.monitoring.complete := FALSE;
   END_IF;
   #_w2 := #_w1 AND #statEnableManualCmds;
   IF #_w2 THEN "Unit1.Em8.ControlNodes".cmThicknessAxisZ.commands.enableAxis := FALSE; END_IF;
   IF #_w2 AND NOT "Unit1.Em8.HmiInterface".cmThicknessAxisZ.monitoring.axisEnabled THEN
       "Unit1.Em8.HmiInterface".cmThicknessAxisZ.commands.enableAxis := TRUE;
   END_IF;
   #_w3 := #_w1 AND NOT #statEnableManualCmds;
   IF #_w3 THEN "Unit1.Em8.HmiInterface".cmThicknessAxisZ.commands.enableAxis := FALSE; END_IF;
   IF #_w3 AND NOT "Unit1.Em8.ControlNodes".cmThicknessAxisZ.monitoring.axisEnabled THEN
       "Unit1.Em8.ControlNodes".cmThicknessAxisZ.commands.enableAxis := TRUE;
   END_IF;
   IF #_w1 AND ("Unit1.Em8.HmiInterface".cmThicknessAxisZ.monitoring.axisEnabled OR "Unit1.Em8.ControlNodes".cmThicknessAxisZ.monitoring.axisEnabled) THEN
       "Unit1.Em8.ControlNodes".cm.brakeTest.thicknessAxisZ.monitoring."step" := 10;
   END_IF;
   "Unit1.Em8.ControlNodes".cm.brakeTest.thicknessAxisZ.commands.brakeSelect := "Unit1.Em8.ControlNodes".cm.brakeTest.thicknessAxisZ.monitoring."step" = 10;
   "Unit1.Em8.ControlNodes".cm.brakeTest.thicknessAxisZ.commands.brakeStart := "Unit1.Em8.ControlNodes".cm.brakeTest.thicknessAxisZ.commands.brakeSelect AND "Unit1.Em8.ControlNodes".cm.brakeTest.thicknessAxisZ.monitoring.brakeSelected;
   #statTonTime[61].TON(IN := "Unit1.Em8.ControlNodes".cm.brakeTest.thicknessAxisZ.commands.brakeSelect AND "Unit1.Em8.ControlNodes".cm.brakeTest.thicknessAxisZ.monitoring.brakeResult AND "Unit1.Em8.ControlNodes".cm.brakeTest.thicknessAxisZ.monitoring.brakeCompleted,
                        PT := T#1ms);
   IF #statTonTime[61].Q THEN
       "Unit1.Em8.ControlNodes".cm.brakeTest.thicknessAxisZ.monitoring."step" := 20;
   END_IF;
   "Unit1.Em8.ControlNodes".cm.brakeTest.thicknessAxisZ.commands.axisReset := "Unit1.Em8.ControlNodes".cm.brakeTest.thicknessAxisZ.monitoring."step" = 20;
   #statTonTime[62].TON(IN := "Unit1.Em8.ControlNodes".cm.brakeTest.thicknessAxisZ.commands.axisReset AND ("Unit1.Em8.ControlNodes".cmThicknessAxisZ.monitoring.resetActive OR "Unit1.Em8.HmiInterface".cmThicknessAxisZ.monitoring.axisEnabled),
                        PT := T#1ms);
   IF #statTonTime[62].Q THEN
       "Unit1.Em8.ControlNodes".cm.brakeTest.thicknessAxisZ.monitoring."step" := 30;
   END_IF;
   #_w4 := "Unit1.Em8.ControlNodes".cm.brakeTest.thicknessAxisZ.monitoring."step" = 30;
   IF #_w4 THEN
       "Unit1.Em8.ControlNodes".cm.brakeTest.thicknessAxisZ.monitoring.busy := FALSE;
       "Unit1.Em8.ControlNodes".cm.brakeTest.thicknessAxisZ.monitoring.complete := TRUE;
   END_IF;
   #statTonTime[63].TON(IN := #_w4, PT := T#1ms);
   IF #statTonTime[63].Q THEN
       "Unit1.Em8.ControlNodes".cm.brakeTest.thicknessAxisZ.monitoring."step" := 0;
   END_IF;
END_REGION

REGION Network 69: Thickness Z-Axis Brake Test Monitoring
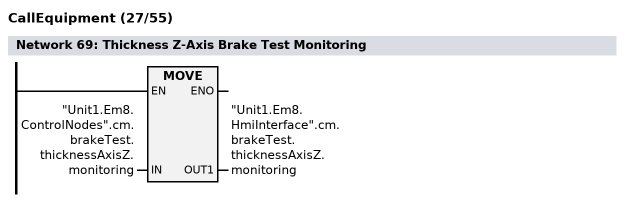
   RUNG wire#powerrail
      Move(in := "Unit1.Em8.ControlNodes".cm.brakeTest.thicknessAxisZ.monitoring, out1 => "Unit1.Em8.HmiInterface".cm.brakeTest.thicknessAxisZ.monitoring)
   END_RUNG
   // the same network as SCL:
   "Unit1.Em8.HmiInterface".cm.brakeTest.thicknessAxisZ.monitoring := "Unit1.Em8.ControlNodes".cm.brakeTest.thicknessAxisZ.monitoring;
END_REGION

REGION Network 70: Call Thickness Z-Axis Telegram 701
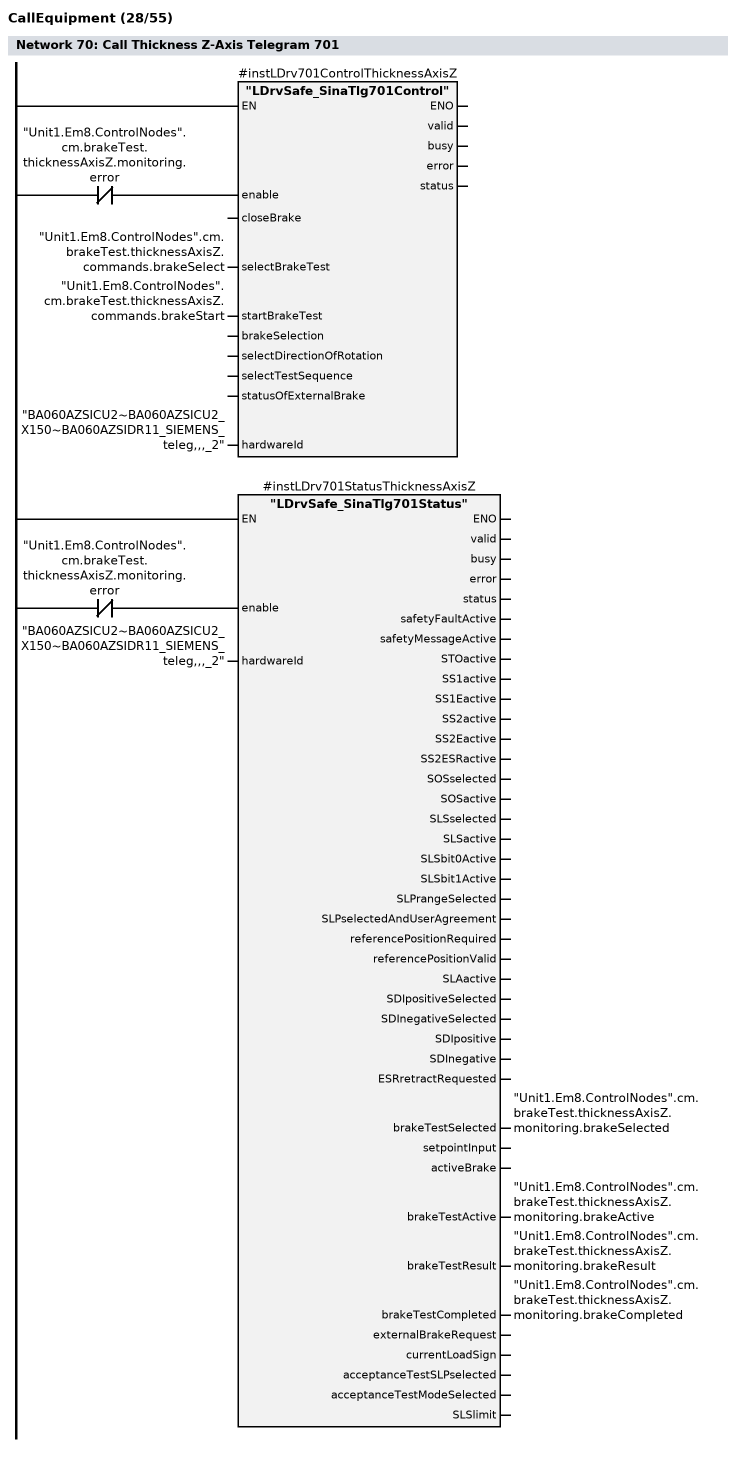
   RUNG wire#powerrail
      #instLDrv701ControlThicknessAxisZ(enable := wire#w1, closeBrake :=, selectBrakeTest := "Unit1.Em8.ControlNodes".cm.brakeTest.thicknessAxisZ.commands.brakeSelect, startBrakeTest := "Unit1.Em8.ControlNodes".cm.brakeTest.thicknessAxisZ.commands.brakeStart, brakeSelection :=, selectDirectionOfRotation :=, selectTestSequence :=, statusOfExternalBrake :=, hardwareId := "BA060AZSICU2~BA060AZSICU2_X150~BA060AZSIDR11_SIEMENS_teleg,,,_2", valid =>, busy =>, error =>, status =>)
   END_RUNG
   RUNG wire#powerrail
      I_Contact( "Unit1.Em8.ControlNodes".cm.brakeTest.thicknessAxisZ.monitoring.error )
   END_RUNG wire#w1
   RUNG wire#powerrail
      #instLDrv701StatusThicknessAxisZ(enable := wire#w2, hardwareId := "BA060AZSICU2~BA060AZSICU2_X150~BA060AZSIDR11_SIEMENS_teleg,,,_2", valid =>, busy =>, error =>, status =>, safetyFaultActive =>, safetyMessageActive =>, STOactive =>, SS1active =>, SS1Eactive =>, SS2active =>, SS2Eactive =>, SS2ESRactive =>, SOSselected =>, SOSactive =>, SLSselected =>, SLSactive =>, SLSbit0Active =>, SLSbit1Active =>, SLPrangeSelected =>, SLPselectedAndUserAgreement =>, referencePositionRequired =>, referencePositionValid =>, SLAactive =>, SDIpositiveSelected =>, SDInegativeSelected =>, SDIpositive =>, SDInegative =>, ESRretractRequested =>, brakeTestSelected => "Unit1.Em8.ControlNodes".cm.brakeTest.thicknessAxisZ.monitoring.brakeSelected, setpointInput =>, activeBrake =>, brakeTestActive => "Unit1.Em8.ControlNodes".cm.brakeTest.thicknessAxisZ.monitoring.brakeActive, brakeTestResult => "Unit1.Em8.ControlNodes".cm.brakeTest.thicknessAxisZ.monitoring.brakeResult, brakeTestCompleted => "Unit1.Em8.ControlNodes".cm.brakeTest.thicknessAxisZ.monitoring.brakeCompleted, externalBrakeRequest =>, currentLoadSign =>, acceptanceTestSLPselected =>, acceptanceTestModeSelected =>, SLSlimit =>)
   END_RUNG
   RUNG wire#powerrail
      I_Contact( "Unit1.Em8.ControlNodes".cm.brakeTest.thicknessAxisZ.monitoring.error )
   END_RUNG wire#w2
   // the same network as SCL:
   #instLDrv701ControlThicknessAxisZ(enable := NOT "Unit1.Em8.ControlNodes".cm.brakeTest.thicknessAxisZ.monitoring.error,   // "LDrvSafe_SinaTlg701Control"
                           selectBrakeTest := "Unit1.Em8.ControlNodes".cm.brakeTest.thicknessAxisZ.commands.brakeSelect,
                           startBrakeTest := "Unit1.Em8.ControlNodes".cm.brakeTest.thicknessAxisZ.commands.brakeStart,
                           hardwareId := "BA060AZSICU2~BA060AZSICU2_X150~BA060AZSIDR11_SIEMENS_teleg,,,_2");
   #instLDrv701StatusThicknessAxisZ(enable := NOT "Unit1.Em8.ControlNodes".cm.brakeTest.thicknessAxisZ.monitoring.error,   // "LDrvSafe_SinaTlg701Status"
                           hardwareId := "BA060AZSICU2~BA060AZSICU2_X150~BA060AZSIDR11_SIEMENS_teleg,,,_2",
                           brakeTestSelected => "Unit1.Em8.ControlNodes".cm.brakeTest.thicknessAxisZ.monitoring.brakeSelected,
                           brakeTestActive => "Unit1.Em8.ControlNodes".cm.brakeTest.thicknessAxisZ.monitoring.brakeActive,
                           brakeTestResult => "Unit1.Em8.ControlNodes".cm.brakeTest.thicknessAxisZ.monitoring.brakeResult,
                           brakeTestCompleted => "Unit1.Em8.ControlNodes".cm.brakeTest.thicknessAxisZ.monitoring.brakeCompleted);
END_REGION

REGION Network 72: ******************** Control Modules (TwoWayActuator) ********************
   // Call control modules that are actuators after the em logic (jobs and sequence), so that the latest commands are applied to the actuators.
END_REGION

REGION Network 73: Reset CMS
   // Reset Axis when the unit is in the resetting state.
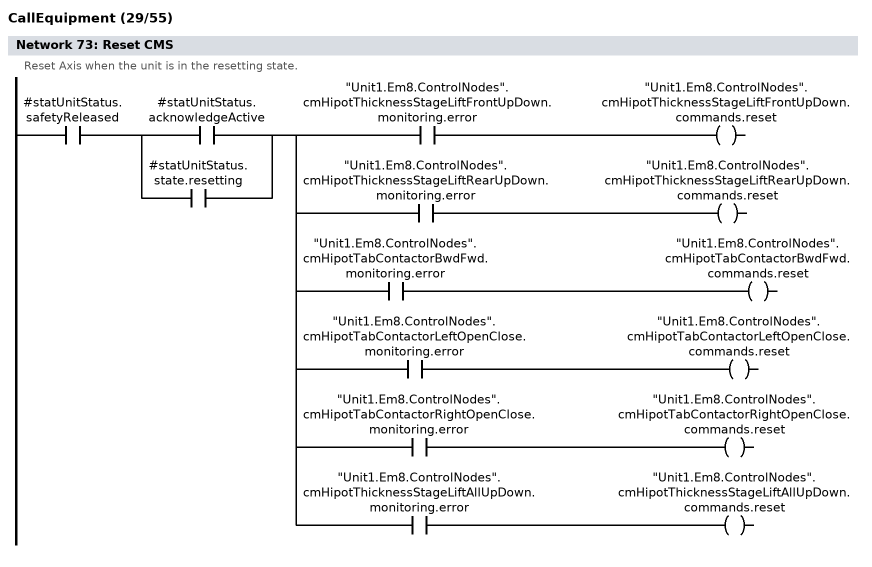
   RUNG wire#powerrail
      Contact( #statUnitStatus.safetyReleased )
      wire#w1
      Contact( #statUnitStatus.acknowledgeActive )
      wire#w2
      Contact( "Unit1.Em8.ControlNodes".cmHipotThicknessStageLiftFrontUpDown.monitoring.error )
      Coil( "Unit1.Em8.ControlNodes".cmHipotThicknessStageLiftFrontUpDown.commands.reset )
   END_RUNG
   RUNG wire#w1
      Contact( #statUnitStatus.state.resetting )
   END_RUNG wire#w2
   RUNG wire#w2
      Contact( "Unit1.Em8.ControlNodes".cmHipotThicknessStageLiftRearUpDown.monitoring.error )
      Coil( "Unit1.Em8.ControlNodes".cmHipotThicknessStageLiftRearUpDown.commands.reset )
   END_RUNG
   RUNG wire#w2
      Contact( "Unit1.Em8.ControlNodes".cmHipotTabContactorBwdFwd.monitoring.error )
      Coil( "Unit1.Em8.ControlNodes".cmHipotTabContactorBwdFwd.commands.reset )
   END_RUNG
   RUNG wire#w2
      Contact( "Unit1.Em8.ControlNodes".cmHipotTabContactorLeftOpenClose.monitoring.error )
      Coil( "Unit1.Em8.ControlNodes".cmHipotTabContactorLeftOpenClose.commands.reset )
   END_RUNG
   RUNG wire#w2
      Contact( "Unit1.Em8.ControlNodes".cmHipotTabContactorRightOpenClose.monitoring.error )
      Coil( "Unit1.Em8.ControlNodes".cmHipotTabContactorRightOpenClose.commands.reset )
   END_RUNG
   RUNG wire#w2
      Contact( "Unit1.Em8.ControlNodes".cmHipotThicknessStageLiftAllUpDown.monitoring.error )
      Coil( "Unit1.Em8.ControlNodes".cmHipotThicknessStageLiftAllUpDown.commands.reset )
   END_RUNG
   // the same network as SCL:
   #_w1 := #statUnitStatus.safetyReleased AND (#statUnitStatus.acknowledgeActive OR #statUnitStatus.state.resetting);
   "Unit1.Em8.ControlNodes".cmHipotThicknessStageLiftFrontUpDown.commands.reset := #_w1 AND "Unit1.Em8.ControlNodes".cmHipotThicknessStageLiftFrontUpDown.monitoring.error;
   "Unit1.Em8.ControlNodes".cmHipotThicknessStageLiftRearUpDown.commands.reset := #_w1 AND "Unit1.Em8.ControlNodes".cmHipotThicknessStageLiftRearUpDown.monitoring.error;
   "Unit1.Em8.ControlNodes".cmHipotTabContactorBwdFwd.commands.reset := #_w1 AND "Unit1.Em8.ControlNodes".cmHipotTabContactorBwdFwd.monitoring.error;
   "Unit1.Em8.ControlNodes".cmHipotTabContactorLeftOpenClose.commands.reset := #_w1 AND "Unit1.Em8.ControlNodes".cmHipotTabContactorLeftOpenClose.monitoring.error;
   "Unit1.Em8.ControlNodes".cmHipotTabContactorRightOpenClose.commands.reset := #_w1 AND "Unit1.Em8.ControlNodes".cmHipotTabContactorRightOpenClose.monitoring.error;
   "Unit1.Em8.ControlNodes".cmHipotThicknessStageLiftAllUpDown.commands.reset := #_w1 AND "Unit1.Em8.ControlNodes".cmHipotThicknessStageLiftAllUpDown.monitoring.error;
END_REGION

REGION Network 75: Hipot & Thickness Stage Lift Front Interlock Condition
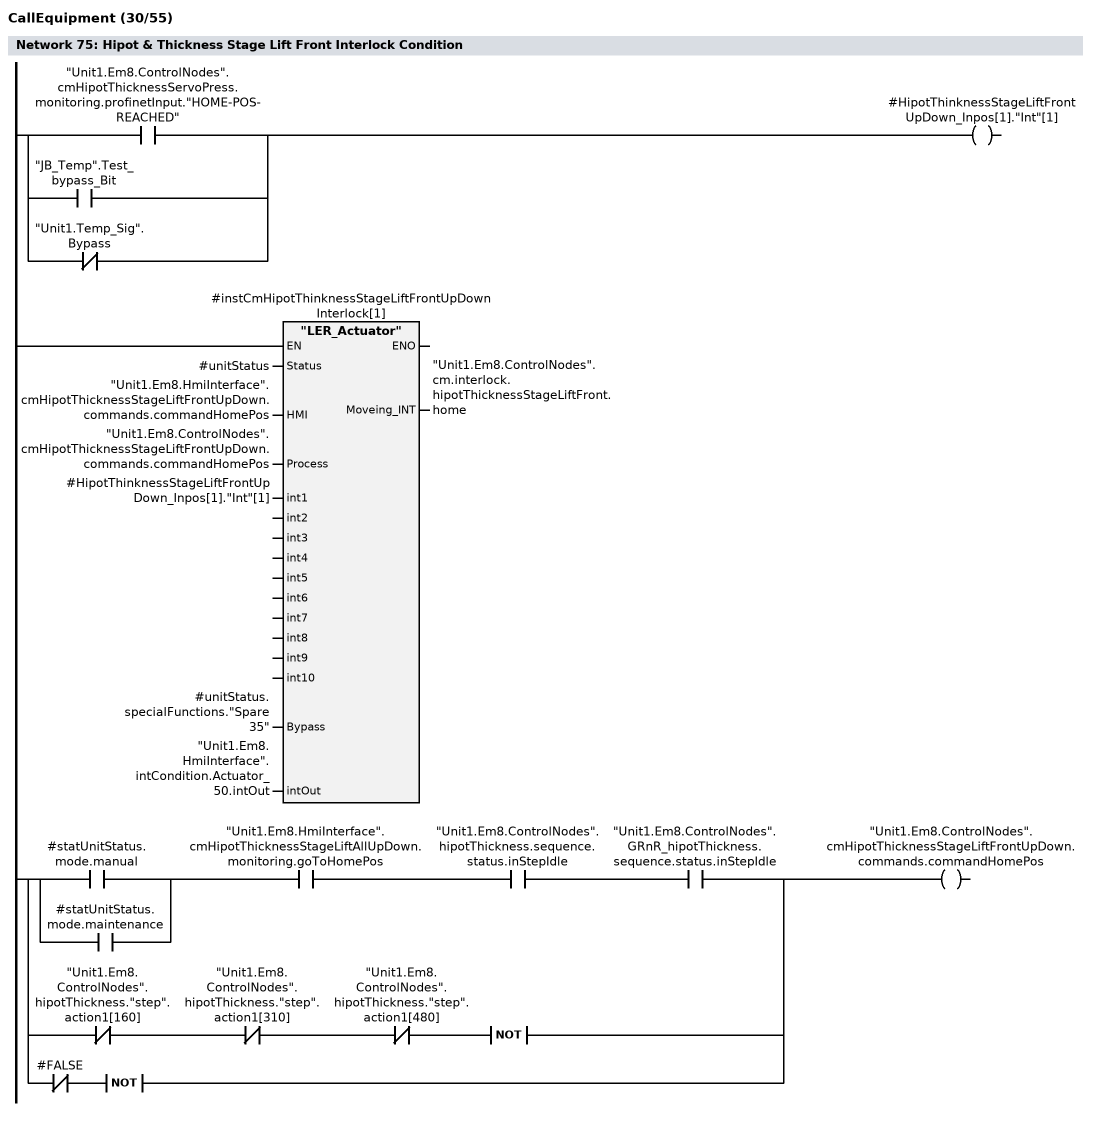
   RUNG wire#powerrail
      Contact( "Unit1.Em8.ControlNodes".cmHipotThicknessServoPress.monitoring.profinetInput."HOME-POS-REACHED" )
      wire#w1
      Coil( #HipotThinknessStageLiftFrontUpDown_Inpos[1]."Int"[1] )
   END_RUNG
   RUNG wire#powerrail
      Contact( "JB_Temp".Test_bypass_Bit )
   END_RUNG wire#w1
   RUNG wire#powerrail
      I_Contact( "Unit1.Temp_Sig".Bypass )
   END_RUNG wire#w1
   RUNG wire#powerrail
      #instCmHipotThinknessStageLiftFrontUpDownInterlock[1](Status := #unitStatus, HMI := "Unit1.Em8.HmiInterface".cmHipotThicknessStageLiftFrontUpDown.commands.commandHomePos, Process := "Unit1.Em8.ControlNodes".cmHipotThicknessStageLiftFrontUpDown.commands.commandHomePos, int1 := #HipotThinknessStageLiftFrontUpDown_Inpos[1]."Int"[1], int2 :=, int3 :=, int4 :=, int5 :=, int6 :=, int7 :=, int8 :=, int9 :=, int10 :=, Bypass := #unitStatus.specialFunctions."Spare 35", intOut := "Unit1.Em8.HmiInterface".intCondition.Actuator_50.intOut, Moveing_INT => "Unit1.Em8.ControlNodes".cm.interlock.hipotThicknessStageLiftFront.home)
   END_RUNG
   RUNG wire#powerrail
      Contact( #statUnitStatus.mode.manual )
      wire#w2
      Contact( "Unit1.Em8.HmiInterface".cmHipotThicknessStageLiftAllUpDown.monitoring.goToHomePos )
      Contact( "Unit1.Em8.ControlNodes".hipotThickness.sequence.status.inStepIdle )
      Contact( "Unit1.Em8.ControlNodes".GRnR_hipotThickness.sequence.status.inStepIdle )
      wire#w3
      Coil( "Unit1.Em8.ControlNodes".cmHipotThicknessStageLiftFrontUpDown.commands.commandHomePos )
   END_RUNG
   RUNG wire#powerrail
      Contact( #statUnitStatus.mode.maintenance )
   END_RUNG wire#w2
   RUNG wire#powerrail
      I_Contact( "Unit1.Em8.ControlNodes".hipotThickness."step".action1[160] )
      I_Contact( "Unit1.Em8.ControlNodes".hipotThickness."step".action1[310] )
      I_Contact( "Unit1.Em8.ControlNodes".hipotThickness."step".action1[480] )
      Not()
   END_RUNG wire#w3
   RUNG wire#powerrail
      I_Contact( #FALSE )
      Not()
   END_RUNG wire#w3
   // the same network as SCL:
   #HipotThinknessStageLiftFrontUpDown_Inpos[1]."Int"[1] := "Unit1.Em8.ControlNodes".cmHipotThicknessServoPress.monitoring.profinetInput."HOME-POS-REACHED" OR "JB_Temp".Test_bypass_Bit OR NOT "Unit1.Temp_Sig".Bypass;
   #instCmHipotThinknessStageLiftFrontUpDownInterlock[1](Status := #unitStatus,   // "LER_Actuator"
                           HMI := "Unit1.Em8.HmiInterface".cmHipotThicknessStageLiftFrontUpDown.commands.commandHomePos,
                           Process := "Unit1.Em8.ControlNodes".cmHipotThicknessStageLiftFrontUpDown.commands.commandHomePos,
                           int1 := #HipotThinknessStageLiftFrontUpDown_Inpos[1]."Int"[1],
                           Bypass := #unitStatus.specialFunctions."Spare 35",
                           intOut := "Unit1.Em8.HmiInterface".intCondition.Actuator_50.intOut,
                           Moveing_INT => "Unit1.Em8.ControlNodes".cm.interlock.hipotThicknessStageLiftFront.home);
   "Unit1.Em8.ControlNodes".cmHipotThicknessStageLiftFrontUpDown.commands.commandHomePos := ((#statUnitStatus.mode.manual OR #statUnitStatus.mode.maintenance) AND "Unit1.Em8.HmiInterface".cmHipotThicknessStageLiftAllUpDown.monitoring.goToHomePos AND "Unit1.Em8.ControlNodes".hipotThickness.sequence.status.inStepIdle AND "Unit1.Em8.ControlNodes".GRnR_hipotThickness.sequence.status.inStepIdle) OR NOT (NOT "Unit1.Em8.ControlNodes".hipotThickness."step".action1[160] AND NOT "Unit1.Em8.ControlNodes".hipotThickness."step".action1[310] AND NOT "Unit1.Em8.ControlNodes".hipotThickness."step".action1[480]) OR NOT (NOT #FALSE);
END_REGION

REGION Network 76: Hipot & Thickness Stage Lift Front Commands
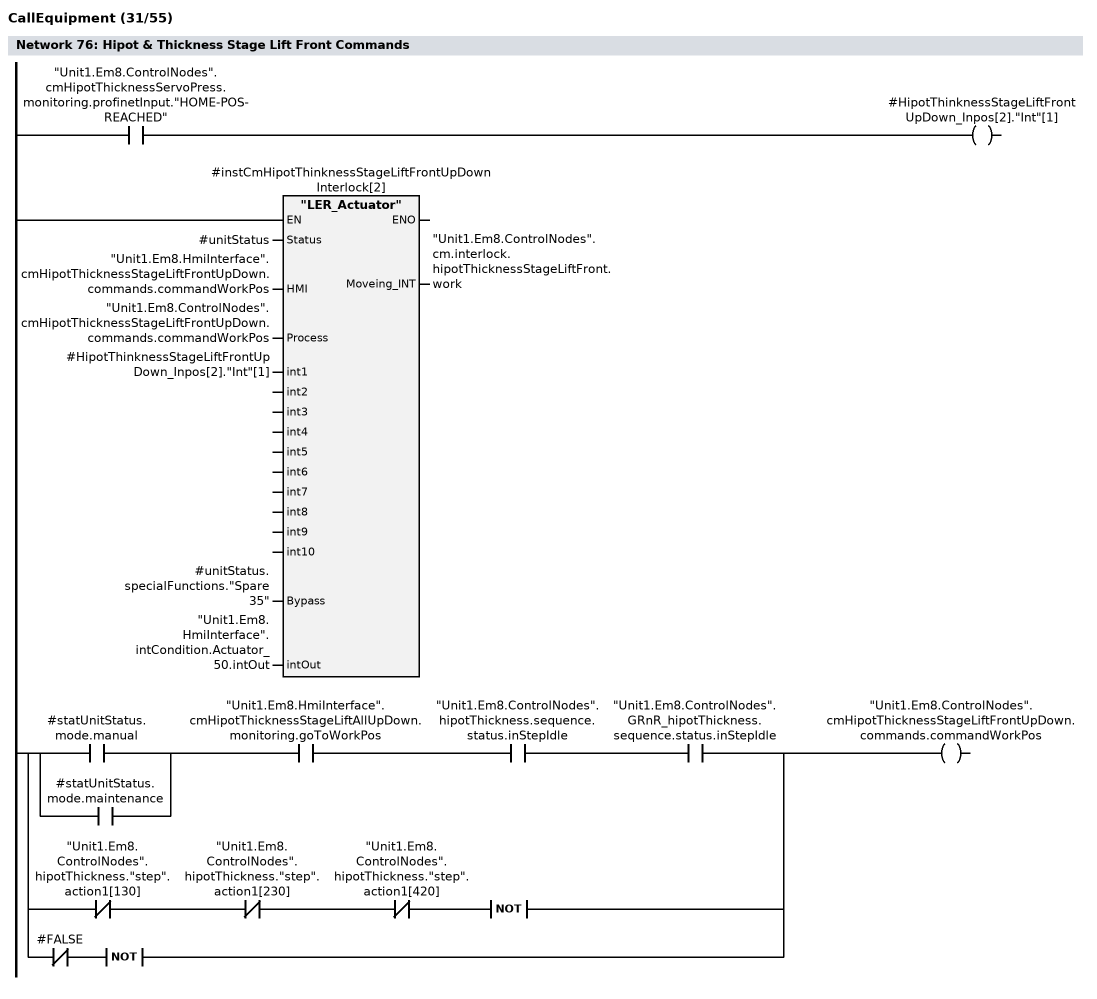
   RUNG wire#powerrail
      Contact( "Unit1.Em8.ControlNodes".cmHipotThicknessServoPress.monitoring.profinetInput."HOME-POS-REACHED" )
      Coil( #HipotThinknessStageLiftFrontUpDown_Inpos[2]."Int"[1] )
   END_RUNG
   RUNG wire#powerrail
      #instCmHipotThinknessStageLiftFrontUpDownInterlock[2](Status := #unitStatus, HMI := "Unit1.Em8.HmiInterface".cmHipotThicknessStageLiftFrontUpDown.commands.commandWorkPos, Process := "Unit1.Em8.ControlNodes".cmHipotThicknessStageLiftFrontUpDown.commands.commandWorkPos, int1 := #HipotThinknessStageLiftFrontUpDown_Inpos[2]."Int"[1], int2 :=, int3 :=, int4 :=, int5 :=, int6 :=, int7 :=, int8 :=, int9 :=, int10 :=, Bypass := #unitStatus.specialFunctions."Spare 35", intOut := "Unit1.Em8.HmiInterface".intCondition.Actuator_50.intOut, Moveing_INT => "Unit1.Em8.ControlNodes".cm.interlock.hipotThicknessStageLiftFront.work)
   END_RUNG
   RUNG wire#powerrail
      Contact( #statUnitStatus.mode.manual )
      wire#w1
      Contact( "Unit1.Em8.HmiInterface".cmHipotThicknessStageLiftAllUpDown.monitoring.goToWorkPos )
      Contact( "Unit1.Em8.ControlNodes".hipotThickness.sequence.status.inStepIdle )
      Contact( "Unit1.Em8.ControlNodes".GRnR_hipotThickness.sequence.status.inStepIdle )
      wire#w2
      Coil( "Unit1.Em8.ControlNodes".cmHipotThicknessStageLiftFrontUpDown.commands.commandWorkPos )
   END_RUNG
   RUNG wire#powerrail
      Contact( #statUnitStatus.mode.maintenance )
   END_RUNG wire#w1
   RUNG wire#powerrail
      I_Contact( "Unit1.Em8.ControlNodes".hipotThickness."step".action1[130] )
      I_Contact( "Unit1.Em8.ControlNodes".hipotThickness."step".action1[230] )
      I_Contact( "Unit1.Em8.ControlNodes".hipotThickness."step".action1[420] )
      Not()
   END_RUNG wire#w2
   RUNG wire#powerrail
      I_Contact( #FALSE )
      Not()
   END_RUNG wire#w2
   // the same network as SCL:
   #HipotThinknessStageLiftFrontUpDown_Inpos[2]."Int"[1] := "Unit1.Em8.ControlNodes".cmHipotThicknessServoPress.monitoring.profinetInput."HOME-POS-REACHED";
   #instCmHipotThinknessStageLiftFrontUpDownInterlock[2](Status := #unitStatus,   // "LER_Actuator"
                           HMI := "Unit1.Em8.HmiInterface".cmHipotThicknessStageLiftFrontUpDown.commands.commandWorkPos,
                           Process := "Unit1.Em8.ControlNodes".cmHipotThicknessStageLiftFrontUpDown.commands.commandWorkPos,
                           int1 := #HipotThinknessStageLiftFrontUpDown_Inpos[2]."Int"[1],
                           Bypass := #unitStatus.specialFunctions."Spare 35",
                           intOut := "Unit1.Em8.HmiInterface".intCondition.Actuator_50.intOut,
                           Moveing_INT => "Unit1.Em8.ControlNodes".cm.interlock.hipotThicknessStageLiftFront.work);
   "Unit1.Em8.ControlNodes".cmHipotThicknessStageLiftFrontUpDown.commands.commandWorkPos := ((#statUnitStatus.mode.manual OR #statUnitStatus.mode.maintenance) AND "Unit1.Em8.HmiInterface".cmHipotThicknessStageLiftAllUpDown.monitoring.goToWorkPos AND "Unit1.Em8.ControlNodes".hipotThickness.sequence.status.inStepIdle AND "Unit1.Em8.ControlNodes".GRnR_hipotThickness.sequence.status.inStepIdle) OR NOT (NOT "Unit1.Em8.ControlNodes".hipotThickness."step".action1[130] AND NOT "Unit1.Em8.ControlNodes".hipotThickness."step".action1[230] AND NOT "Unit1.Em8.ControlNodes".hipotThickness."step".action1[420]) OR NOT (NOT #FALSE);
END_REGION

REGION Network 77: Call CM Hipot & Thickness Stage Lift Front Cylinder Up/Down (LBC_TwoWayActuator)
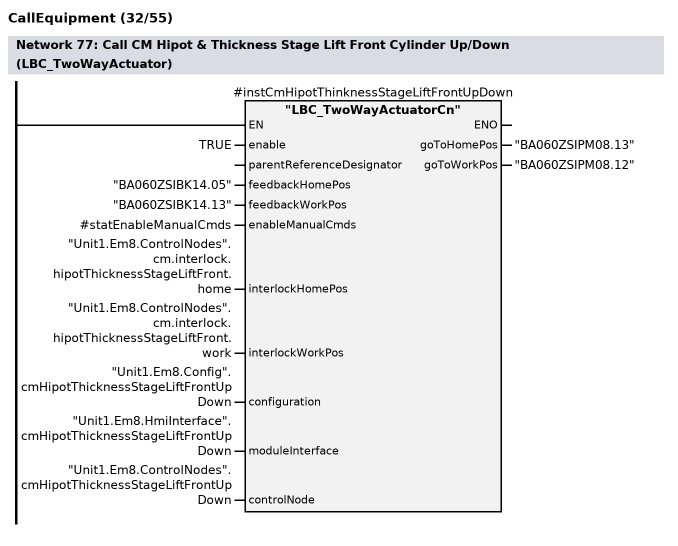
   RUNG wire#powerrail
      #instCmHipotThinknessStageLiftFrontUpDown(enable := TRUE, parentReferenceDesignator :=, feedbackHomePos := "BA060ZSIBK14.05", feedbackWorkPos := "BA060ZSIBK14.13", enableManualCmds := #statEnableManualCmds, interlockHomePos := "Unit1.Em8.ControlNodes".cm.interlock.hipotThicknessStageLiftFront.home, interlockWorkPos := "Unit1.Em8.ControlNodes".cm.interlock.hipotThicknessStageLiftFront.work, configuration := "Unit1.Em8.Config".cmHipotThicknessStageLiftFrontUpDown, moduleInterface := "Unit1.Em8.HmiInterface".cmHipotThicknessStageLiftFrontUpDown, controlNode := "Unit1.Em8.ControlNodes".cmHipotThicknessStageLiftFrontUpDown, goToHomePos => "BA060ZSIPM08.13", goToWorkPos => "BA060ZSIPM08.12")
   END_RUNG
   // the same network as SCL:
   #instCmHipotThinknessStageLiftFrontUpDown(enable := TRUE,   // "LBC_TwoWayActuatorCn"
                           feedbackHomePos := "BA060ZSIBK14.05",
                           feedbackWorkPos := "BA060ZSIBK14.13",
                           enableManualCmds := #statEnableManualCmds,
                           interlockHomePos := "Unit1.Em8.ControlNodes".cm.interlock.hipotThicknessStageLiftFront.home,
                           interlockWorkPos := "Unit1.Em8.ControlNodes".cm.interlock.hipotThicknessStageLiftFront.work,
                           configuration := "Unit1.Em8.Config".cmHipotThicknessStageLiftFrontUpDown,
                           moduleInterface := "Unit1.Em8.HmiInterface".cmHipotThicknessStageLiftFrontUpDown,
                           controlNode := "Unit1.Em8.ControlNodes".cmHipotThicknessStageLiftFrontUpDown,
                           goToHomePos => "BA060ZSIPM08.13",
                           goToWorkPos => "BA060ZSIPM08.12");
END_REGION

REGION Network 79: Hipot & Thickness Stage Lift Rear Interlock Condition
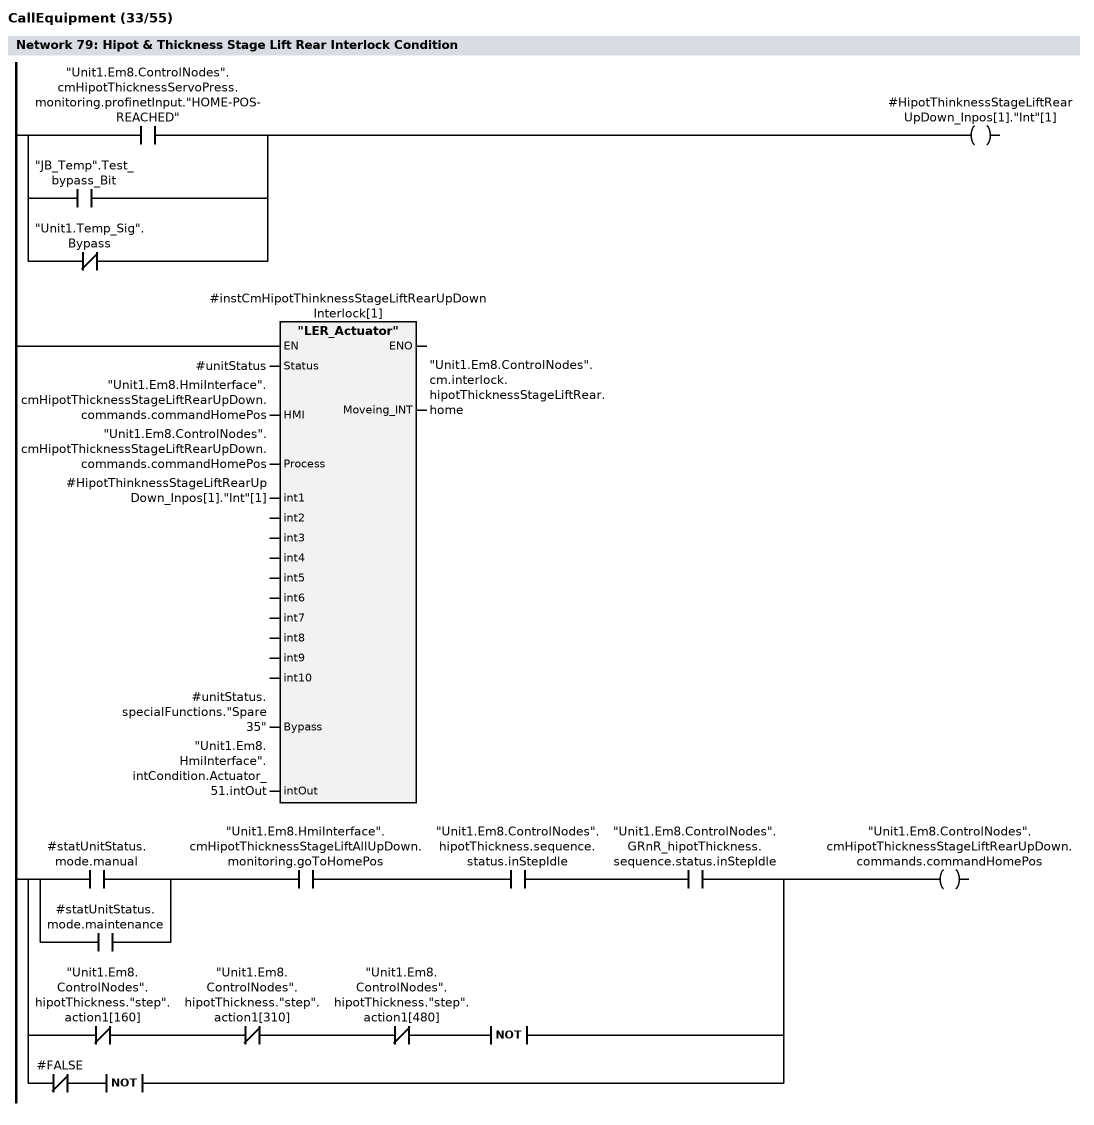
   RUNG wire#powerrail
      Contact( "Unit1.Em8.ControlNodes".cmHipotThicknessServoPress.monitoring.profinetInput."HOME-POS-REACHED" )
      wire#w1
      Coil( #HipotThinknessStageLiftRearUpDown_Inpos[1]."Int"[1] )
   END_RUNG
   RUNG wire#powerrail
      Contact( "JB_Temp".Test_bypass_Bit )
   END_RUNG wire#w1
   RUNG wire#powerrail
      I_Contact( "Unit1.Temp_Sig".Bypass )
   END_RUNG wire#w1
   RUNG wire#powerrail
      #instCmHipotThinknessStageLiftRearUpDownInterlock[1](Status := #unitStatus, HMI := "Unit1.Em8.HmiInterface".cmHipotThicknessStageLiftRearUpDown.commands.commandHomePos, Process := "Unit1.Em8.ControlNodes".cmHipotThicknessStageLiftRearUpDown.commands.commandHomePos, int1 := #HipotThinknessStageLiftRearUpDown_Inpos[1]."Int"[1], int2 :=, int3 :=, int4 :=, int5 :=, int6 :=, int7 :=, int8 :=, int9 :=, int10 :=, Bypass := #unitStatus.specialFunctions."Spare 35", intOut := "Unit1.Em8.HmiInterface".intCondition.Actuator_51.intOut, Moveing_INT => "Unit1.Em8.ControlNodes".cm.interlock.hipotThicknessStageLiftRear.home)
   END_RUNG
   RUNG wire#powerrail
      Contact( #statUnitStatus.mode.manual )
      wire#w2
      Contact( "Unit1.Em8.HmiInterface".cmHipotThicknessStageLiftAllUpDown.monitoring.goToHomePos )
      Contact( "Unit1.Em8.ControlNodes".hipotThickness.sequence.status.inStepIdle )
      Contact( "Unit1.Em8.ControlNodes".GRnR_hipotThickness.sequence.status.inStepIdle )
      wire#w3
      Coil( "Unit1.Em8.ControlNodes".cmHipotThicknessStageLiftRearUpDown.commands.commandHomePos )
   END_RUNG
   RUNG wire#powerrail
      Contact( #statUnitStatus.mode.maintenance )
   END_RUNG wire#w2
   RUNG wire#powerrail
      I_Contact( "Unit1.Em8.ControlNodes".hipotThickness."step".action1[160] )
      I_Contact( "Unit1.Em8.ControlNodes".hipotThickness."step".action1[310] )
      I_Contact( "Unit1.Em8.ControlNodes".hipotThickness."step".action1[480] )
      Not()
   END_RUNG wire#w3
   RUNG wire#powerrail
      I_Contact( #FALSE )
      Not()
   END_RUNG wire#w3
   // the same network as SCL:
   #HipotThinknessStageLiftRearUpDown_Inpos[1]."Int"[1] := "Unit1.Em8.ControlNodes".cmHipotThicknessServoPress.monitoring.profinetInput."HOME-POS-REACHED" OR "JB_Temp".Test_bypass_Bit OR NOT "Unit1.Temp_Sig".Bypass;
   #instCmHipotThinknessStageLiftRearUpDownInterlock[1](Status := #unitStatus,   // "LER_Actuator"
                           HMI := "Unit1.Em8.HmiInterface".cmHipotThicknessStageLiftRearUpDown.commands.commandHomePos,
                           Process := "Unit1.Em8.ControlNodes".cmHipotThicknessStageLiftRearUpDown.commands.commandHomePos,
                           int1 := #HipotThinknessStageLiftRearUpDown_Inpos[1]."Int"[1],
                           Bypass := #unitStatus.specialFunctions."Spare 35",
                           intOut := "Unit1.Em8.HmiInterface".intCondition.Actuator_51.intOut,
                           Moveing_INT => "Unit1.Em8.ControlNodes".cm.interlock.hipotThicknessStageLiftRear.home);
   "Unit1.Em8.ControlNodes".cmHipotThicknessStageLiftRearUpDown.commands.commandHomePos := ((#statUnitStatus.mode.manual OR #statUnitStatus.mode.maintenance) AND "Unit1.Em8.HmiInterface".cmHipotThicknessStageLiftAllUpDown.monitoring.goToHomePos AND "Unit1.Em8.ControlNodes".hipotThickness.sequence.status.inStepIdle AND "Unit1.Em8.ControlNodes".GRnR_hipotThickness.sequence.status.inStepIdle) OR NOT (NOT "Unit1.Em8.ControlNodes".hipotThickness."step".action1[160] AND NOT "Unit1.Em8.ControlNodes".hipotThickness."step".action1[310] AND NOT "Unit1.Em8.ControlNodes".hipotThickness."step".action1[480]) OR NOT (NOT #FALSE);
END_REGION

REGION Network 80: Hipot & Thickness Stage Lift Rear Commands
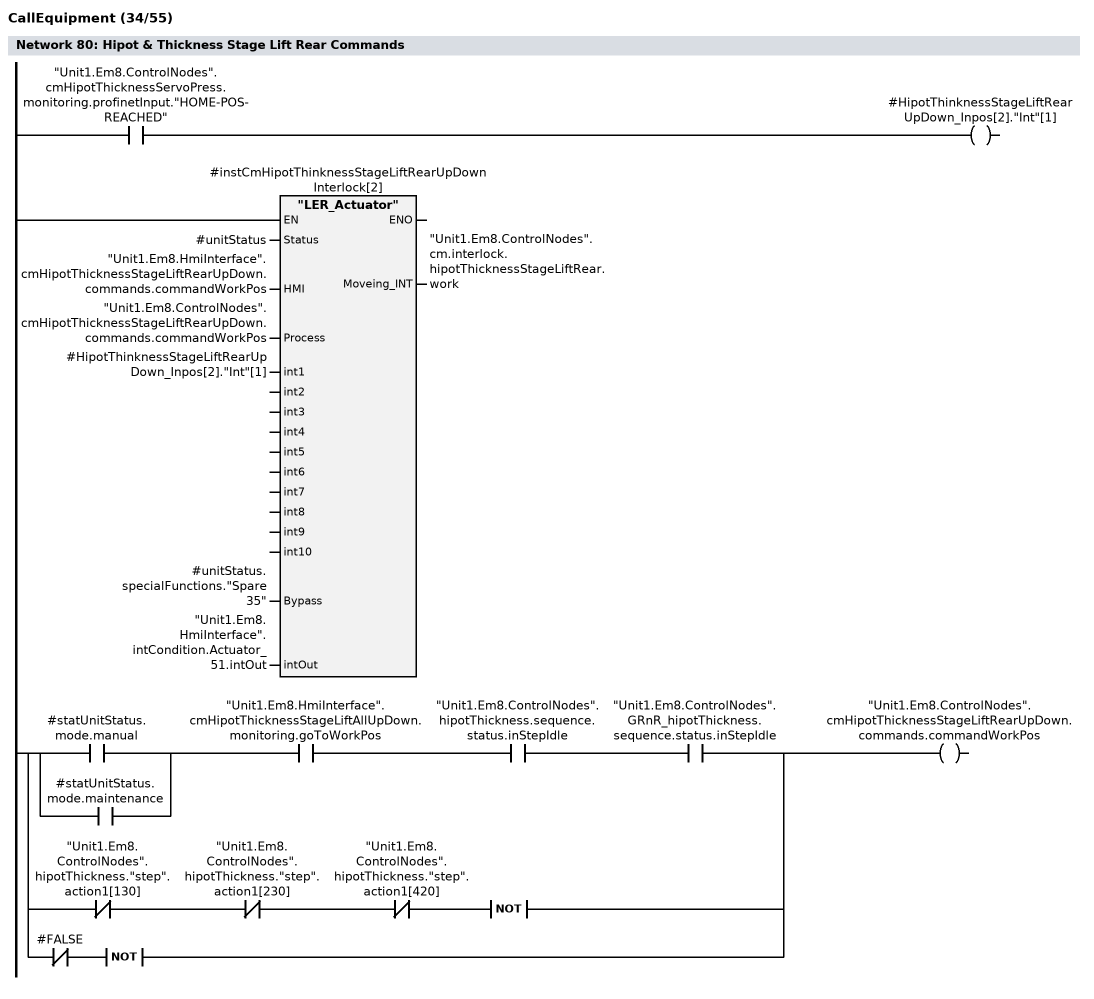
   RUNG wire#powerrail
      Contact( "Unit1.Em8.ControlNodes".cmHipotThicknessServoPress.monitoring.profinetInput."HOME-POS-REACHED" )
      Coil( #HipotThinknessStageLiftRearUpDown_Inpos[2]."Int"[1] )
   END_RUNG
   RUNG wire#powerrail
      #instCmHipotThinknessStageLiftRearUpDownInterlock[2](Status := #unitStatus, HMI := "Unit1.Em8.HmiInterface".cmHipotThicknessStageLiftRearUpDown.commands.commandWorkPos, Process := "Unit1.Em8.ControlNodes".cmHipotThicknessStageLiftRearUpDown.commands.commandWorkPos, int1 := #HipotThinknessStageLiftRearUpDown_Inpos[2]."Int"[1], int2 :=, int3 :=, int4 :=, int5 :=, int6 :=, int7 :=, int8 :=, int9 :=, int10 :=, Bypass := #unitStatus.specialFunctions."Spare 35", intOut := "Unit1.Em8.HmiInterface".intCondition.Actuator_51.intOut, Moveing_INT => "Unit1.Em8.ControlNodes".cm.interlock.hipotThicknessStageLiftRear.work)
   END_RUNG
   RUNG wire#powerrail
      Contact( #statUnitStatus.mode.manual )
      wire#w1
      Contact( "Unit1.Em8.HmiInterface".cmHipotThicknessStageLiftAllUpDown.monitoring.goToWorkPos )
      Contact( "Unit1.Em8.ControlNodes".hipotThickness.sequence.status.inStepIdle )
      Contact( "Unit1.Em8.ControlNodes".GRnR_hipotThickness.sequence.status.inStepIdle )
      wire#w2
      Coil( "Unit1.Em8.ControlNodes".cmHipotThicknessStageLiftRearUpDown.commands.commandWorkPos )
   END_RUNG
   RUNG wire#powerrail
      Contact( #statUnitStatus.mode.maintenance )
   END_RUNG wire#w1
   RUNG wire#powerrail
      I_Contact( "Unit1.Em8.ControlNodes".hipotThickness."step".action1[130] )
      I_Contact( "Unit1.Em8.ControlNodes".hipotThickness."step".action1[230] )
      I_Contact( "Unit1.Em8.ControlNodes".hipotThickness."step".action1[420] )
      Not()
   END_RUNG wire#w2
   RUNG wire#powerrail
      I_Contact( #FALSE )
      Not()
   END_RUNG wire#w2
   // the same network as SCL:
   #HipotThinknessStageLiftRearUpDown_Inpos[2]."Int"[1] := "Unit1.Em8.ControlNodes".cmHipotThicknessServoPress.monitoring.profinetInput."HOME-POS-REACHED";
   #instCmHipotThinknessStageLiftRearUpDownInterlock[2](Status := #unitStatus,   // "LER_Actuator"
                           HMI := "Unit1.Em8.HmiInterface".cmHipotThicknessStageLiftRearUpDown.commands.commandWorkPos,
                           Process := "Unit1.Em8.ControlNodes".cmHipotThicknessStageLiftRearUpDown.commands.commandWorkPos,
                           int1 := #HipotThinknessStageLiftRearUpDown_Inpos[2]."Int"[1],
                           Bypass := #unitStatus.specialFunctions."Spare 35",
                           intOut := "Unit1.Em8.HmiInterface".intCondition.Actuator_51.intOut,
                           Moveing_INT => "Unit1.Em8.ControlNodes".cm.interlock.hipotThicknessStageLiftRear.work);
   "Unit1.Em8.ControlNodes".cmHipotThicknessStageLiftRearUpDown.commands.commandWorkPos := ((#statUnitStatus.mode.manual OR #statUnitStatus.mode.maintenance) AND "Unit1.Em8.HmiInterface".cmHipotThicknessStageLiftAllUpDown.monitoring.goToWorkPos AND "Unit1.Em8.ControlNodes".hipotThickness.sequence.status.inStepIdle AND "Unit1.Em8.ControlNodes".GRnR_hipotThickness.sequence.status.inStepIdle) OR NOT (NOT "Unit1.Em8.ControlNodes".hipotThickness."step".action1[130] AND NOT "Unit1.Em8.ControlNodes".hipotThickness."step".action1[230] AND NOT "Unit1.Em8.ControlNodes".hipotThickness."step".action1[420]) OR NOT (NOT #FALSE);
END_REGION

REGION Network 81: Call CM Hipot & Thickness Stage Lift Rear Up/Down (LBC_TwoWayActuator)
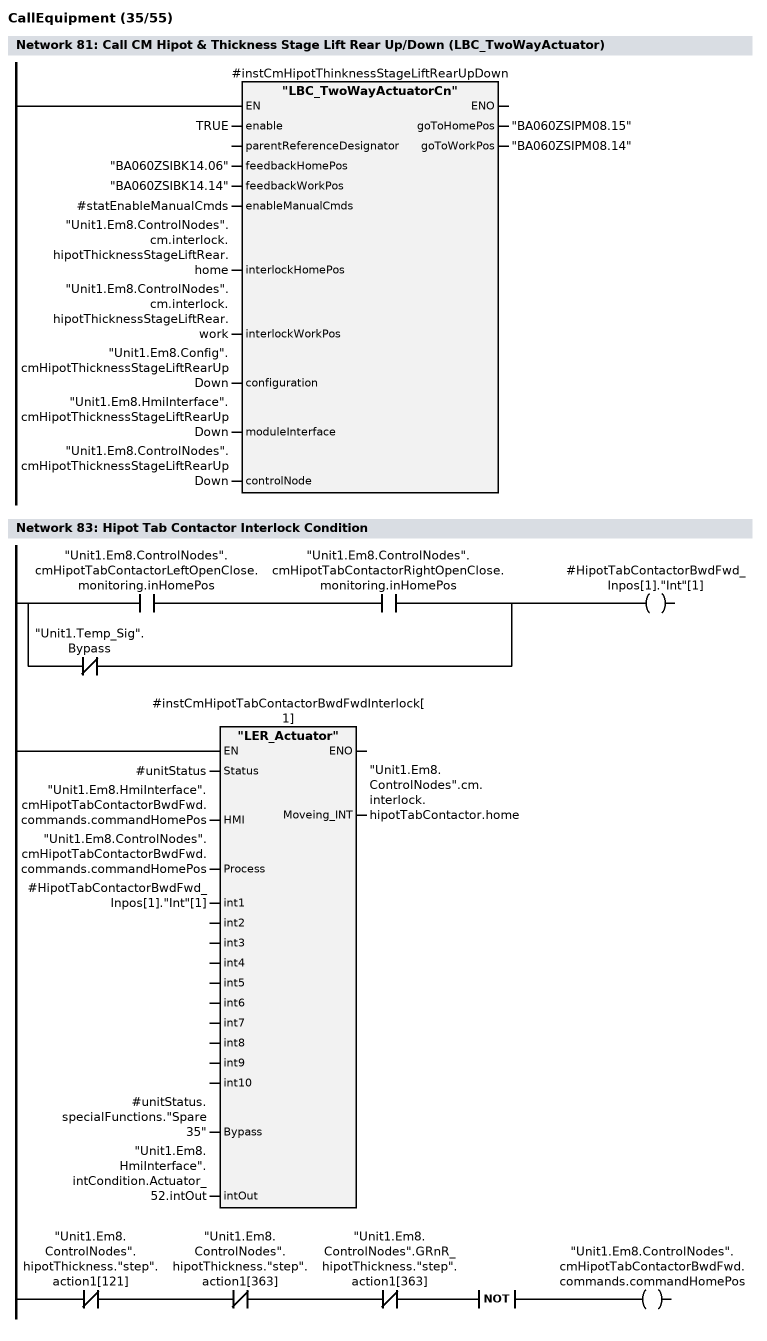
   RUNG wire#powerrail
      #instCmHipotThinknessStageLiftRearUpDown(enable := TRUE, parentReferenceDesignator :=, feedbackHomePos := "BA060ZSIBK14.06", feedbackWorkPos := "BA060ZSIBK14.14", enableManualCmds := #statEnableManualCmds, interlockHomePos := "Unit1.Em8.ControlNodes".cm.interlock.hipotThicknessStageLiftRear.home, interlockWorkPos := "Unit1.Em8.ControlNodes".cm.interlock.hipotThicknessStageLiftRear.work, configuration := "Unit1.Em8.Config".cmHipotThicknessStageLiftRearUpDown, moduleInterface := "Unit1.Em8.HmiInterface".cmHipotThicknessStageLiftRearUpDown, controlNode := "Unit1.Em8.ControlNodes".cmHipotThicknessStageLiftRearUpDown, goToHomePos => "BA060ZSIPM08.15", goToWorkPos => "BA060ZSIPM08.14")
   END_RUNG
   // the same network as SCL:
   #instCmHipotThinknessStageLiftRearUpDown(enable := TRUE,   // "LBC_TwoWayActuatorCn"
                           feedbackHomePos := "BA060ZSIBK14.06",
                           feedbackWorkPos := "BA060ZSIBK14.14",
                           enableManualCmds := #statEnableManualCmds,
                           interlockHomePos := "Unit1.Em8.ControlNodes".cm.interlock.hipotThicknessStageLiftRear.home,
                           interlockWorkPos := "Unit1.Em8.ControlNodes".cm.interlock.hipotThicknessStageLiftRear.work,
                           configuration := "Unit1.Em8.Config".cmHipotThicknessStageLiftRearUpDown,
                           moduleInterface := "Unit1.Em8.HmiInterface".cmHipotThicknessStageLiftRearUpDown,
                           controlNode := "Unit1.Em8.ControlNodes".cmHipotThicknessStageLiftRearUpDown,
                           goToHomePos => "BA060ZSIPM08.15",
                           goToWorkPos => "BA060ZSIPM08.14");
END_REGION

REGION Network 83: Hipot Tab Contactor Interlock Condition
   RUNG wire#powerrail
      Contact( "Unit1.Em8.ControlNodes".cmHipotTabContactorLeftOpenClose.monitoring.inHomePos )
      Contact( "Unit1.Em8.ControlNodes".cmHipotTabContactorRightOpenClose.monitoring.inHomePos )
      wire#w1
      Coil( #HipotTabContactorBwdFwd_Inpos[1]."Int"[1] )
   END_RUNG
   RUNG wire#powerrail
      I_Contact( "Unit1.Temp_Sig".Bypass )
   END_RUNG wire#w1
   RUNG wire#powerrail
      #instCmHipotTabContactorBwdFwdInterlock[1](Status := #unitStatus, HMI := "Unit1.Em8.HmiInterface".cmHipotTabContactorBwdFwd.commands.commandHomePos, Process := "Unit1.Em8.ControlNodes".cmHipotTabContactorBwdFwd.commands.commandHomePos, int1 := #HipotTabContactorBwdFwd_Inpos[1]."Int"[1], int2 :=, int3 :=, int4 :=, int5 :=, int6 :=, int7 :=, int8 :=, int9 :=, int10 :=, Bypass := #unitStatus.specialFunctions."Spare 35", intOut := "Unit1.Em8.HmiInterface".intCondition.Actuator_52.intOut, Moveing_INT => "Unit1.Em8.ControlNodes".cm.interlock.hipotTabContactor.home)
   END_RUNG
   RUNG wire#powerrail
      I_Contact( "Unit1.Em8.ControlNodes".hipotThickness."step".action1[121] )
      I_Contact( "Unit1.Em8.ControlNodes".hipotThickness."step".action1[363] )
      I_Contact( "Unit1.Em8.ControlNodes".GRnR_hipotThickness."step".action1[363] )
      Not()
      Coil( "Unit1.Em8.ControlNodes".cmHipotTabContactorBwdFwd.commands.commandHomePos )
   END_RUNG
   // the same network as SCL:
   #HipotTabContactorBwdFwd_Inpos[1]."Int"[1] := ("Unit1.Em8.ControlNodes".cmHipotTabContactorLeftOpenClose.monitoring.inHomePos AND "Unit1.Em8.ControlNodes".cmHipotTabContactorRightOpenClose.monitoring.inHomePos) OR NOT "Unit1.Temp_Sig".Bypass;
   #instCmHipotTabContactorBwdFwdInterlock[1](Status := #unitStatus,   // "LER_Actuator"
                           HMI := "Unit1.Em8.HmiInterface".cmHipotTabContactorBwdFwd.commands.commandHomePos,
                           Process := "Unit1.Em8.ControlNodes".cmHipotTabContactorBwdFwd.commands.commandHomePos,
                           int1 := #HipotTabContactorBwdFwd_Inpos[1]."Int"[1],
                           Bypass := #unitStatus.specialFunctions."Spare 35",
                           intOut := "Unit1.Em8.HmiInterface".intCondition.Actuator_52.intOut,
                           Moveing_INT => "Unit1.Em8.ControlNodes".cm.interlock.hipotTabContactor.home);
   "Unit1.Em8.ControlNodes".cmHipotTabContactorBwdFwd.commands.commandHomePos := NOT (NOT "Unit1.Em8.ControlNodes".hipotThickness."step".action1[121] AND NOT "Unit1.Em8.ControlNodes".hipotThickness."step".action1[363] AND NOT "Unit1.Em8.ControlNodes".GRnR_hipotThickness."step".action1[363]);
END_REGION

REGION Network 84: Hipot Tab Contactor Commands
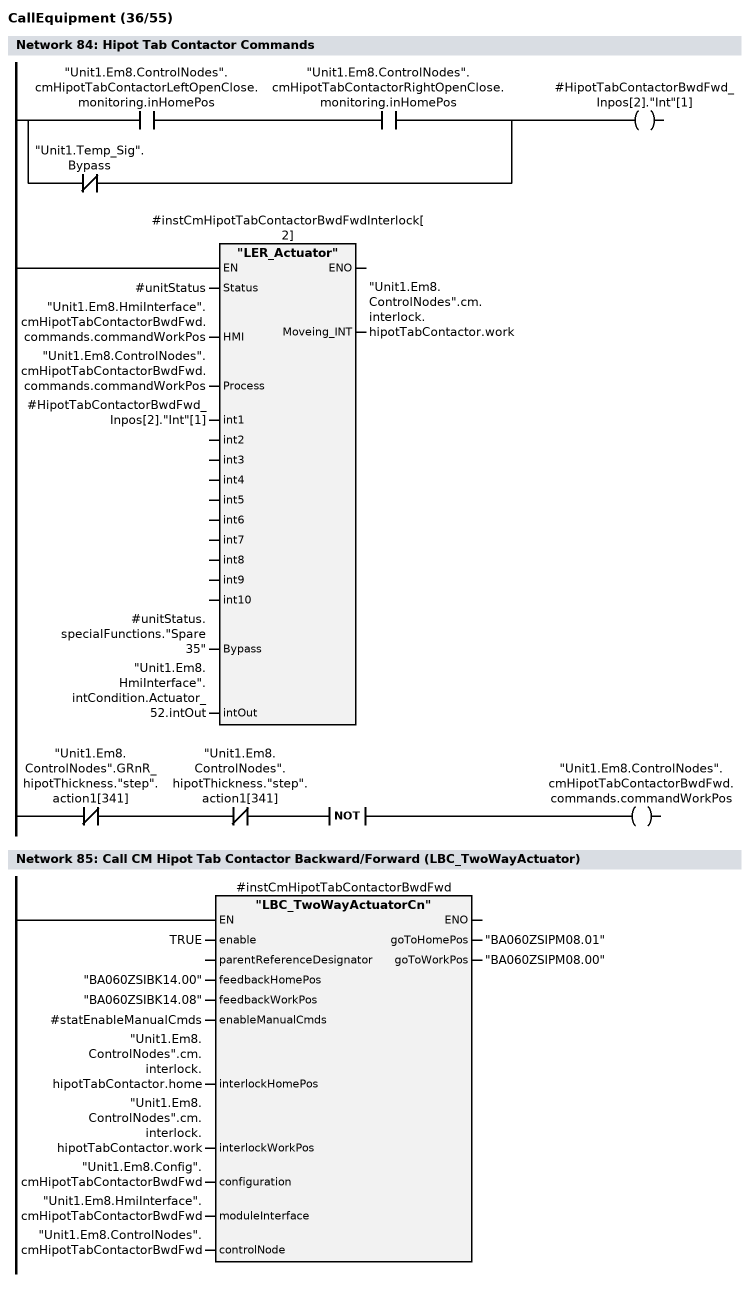
   RUNG wire#powerrail
      Contact( "Unit1.Em8.ControlNodes".cmHipotTabContactorLeftOpenClose.monitoring.inHomePos )
      Contact( "Unit1.Em8.ControlNodes".cmHipotTabContactorRightOpenClose.monitoring.inHomePos )
      wire#w1
      Coil( #HipotTabContactorBwdFwd_Inpos[2]."Int"[1] )
   END_RUNG
   RUNG wire#powerrail
      I_Contact( "Unit1.Temp_Sig".Bypass )
   END_RUNG wire#w1
   RUNG wire#powerrail
      #instCmHipotTabContactorBwdFwdInterlock[2](Status := #unitStatus, HMI := "Unit1.Em8.HmiInterface".cmHipotTabContactorBwdFwd.commands.commandWorkPos, Process := "Unit1.Em8.ControlNodes".cmHipotTabContactorBwdFwd.commands.commandWorkPos, int1 := #HipotTabContactorBwdFwd_Inpos[2]."Int"[1], int2 :=, int3 :=, int4 :=, int5 :=, int6 :=, int7 :=, int8 :=, int9 :=, int10 :=, Bypass := #unitStatus.specialFunctions."Spare 35", intOut := "Unit1.Em8.HmiInterface".intCondition.Actuator_52.intOut, Moveing_INT => "Unit1.Em8.ControlNodes".cm.interlock.hipotTabContactor.work)
   END_RUNG
   RUNG wire#powerrail
      I_Contact( "Unit1.Em8.ControlNodes".GRnR_hipotThickness."step".action1[341] )
      I_Contact( "Unit1.Em8.ControlNodes".hipotThickness."step".action1[341] )
      Not()
      Coil( "Unit1.Em8.ControlNodes".cmHipotTabContactorBwdFwd.commands.commandWorkPos )
   END_RUNG
   // the same network as SCL:
   #HipotTabContactorBwdFwd_Inpos[2]."Int"[1] := ("Unit1.Em8.ControlNodes".cmHipotTabContactorLeftOpenClose.monitoring.inHomePos AND "Unit1.Em8.ControlNodes".cmHipotTabContactorRightOpenClose.monitoring.inHomePos) OR NOT "Unit1.Temp_Sig".Bypass;
   #instCmHipotTabContactorBwdFwdInterlock[2](Status := #unitStatus,   // "LER_Actuator"
                           HMI := "Unit1.Em8.HmiInterface".cmHipotTabContactorBwdFwd.commands.commandWorkPos,
                           Process := "Unit1.Em8.ControlNodes".cmHipotTabContactorBwdFwd.commands.commandWorkPos,
                           int1 := #HipotTabContactorBwdFwd_Inpos[2]."Int"[1],
                           Bypass := #unitStatus.specialFunctions."Spare 35",
                           intOut := "Unit1.Em8.HmiInterface".intCondition.Actuator_52.intOut,
                           Moveing_INT => "Unit1.Em8.ControlNodes".cm.interlock.hipotTabContactor.work);
   "Unit1.Em8.ControlNodes".cmHipotTabContactorBwdFwd.commands.commandWorkPos := NOT (NOT "Unit1.Em8.ControlNodes".GRnR_hipotThickness."step".action1[341] AND NOT "Unit1.Em8.ControlNodes".hipotThickness."step".action1[341]);
END_REGION

REGION Network 85: Call CM Hipot Tab Contactor Backward/Forward (LBC_TwoWayActuator)
   RUNG wire#powerrail
      #instCmHipotTabContactorBwdFwd(enable := TRUE, parentReferenceDesignator :=, feedbackHomePos := "BA060ZSIBK14.00", feedbackWorkPos := "BA060ZSIBK14.08", enableManualCmds := #statEnableManualCmds, interlockHomePos := "Unit1.Em8.ControlNodes".cm.interlock.hipotTabContactor.home, interlockWorkPos := "Unit1.Em8.ControlNodes".cm.interlock.hipotTabContactor.work, configuration := "Unit1.Em8.Config".cmHipotTabContactorBwdFwd, moduleInterface := "Unit1.Em8.HmiInterface".cmHipotTabContactorBwdFwd, controlNode := "Unit1.Em8.ControlNodes".cmHipotTabContactorBwdFwd, goToHomePos => "BA060ZSIPM08.01", goToWorkPos => "BA060ZSIPM08.00")
   END_RUNG
   // the same network as SCL:
   #instCmHipotTabContactorBwdFwd(enable := TRUE,   // "LBC_TwoWayActuatorCn"
                           feedbackHomePos := "BA060ZSIBK14.00",
                           feedbackWorkPos := "BA060ZSIBK14.08",
                           enableManualCmds := #statEnableManualCmds,
                           interlockHomePos := "Unit1.Em8.ControlNodes".cm.interlock.hipotTabContactor.home,
                           interlockWorkPos := "Unit1.Em8.ControlNodes".cm.interlock.hipotTabContactor.work,
                           configuration := "Unit1.Em8.Config".cmHipotTabContactorBwdFwd,
                           moduleInterface := "Unit1.Em8.HmiInterface".cmHipotTabContactorBwdFwd,
                           controlNode := "Unit1.Em8.ControlNodes".cmHipotTabContactorBwdFwd,
                           goToHomePos => "BA060ZSIPM08.01",
                           goToWorkPos => "BA060ZSIPM08.00");
END_REGION

REGION Network 87: Hipot Tab Contactor Left Interlock Condition
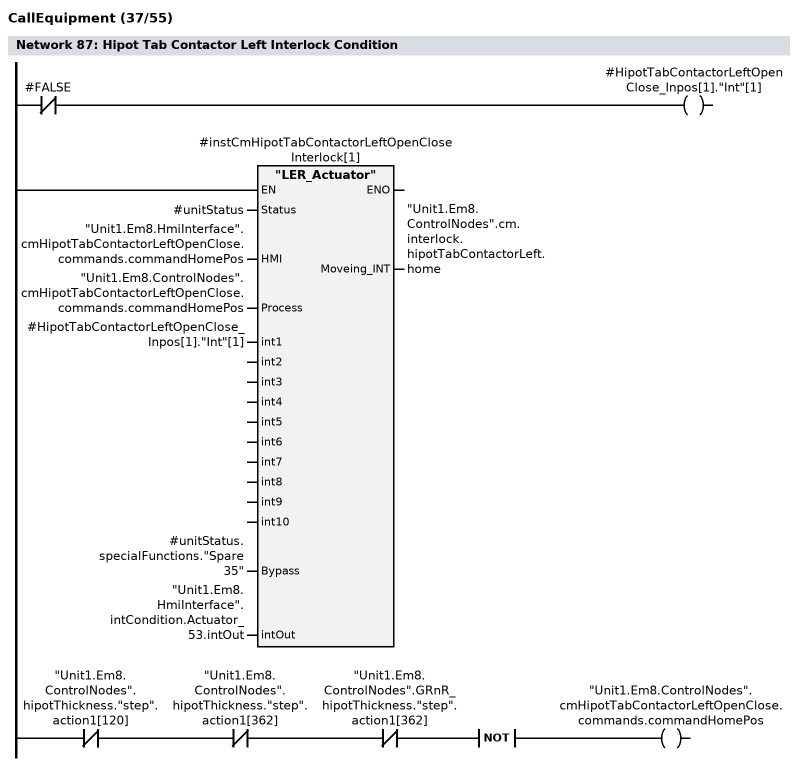
   RUNG wire#powerrail
      I_Contact( #FALSE )
      Coil( #HipotTabContactorLeftOpenClose_Inpos[1]."Int"[1] )
   END_RUNG
   RUNG wire#powerrail
      #instCmHipotTabContactorLeftOpenCloseInterlock[1](Status := #unitStatus, HMI := "Unit1.Em8.HmiInterface".cmHipotTabContactorLeftOpenClose.commands.commandHomePos, Process := "Unit1.Em8.ControlNodes".cmHipotTabContactorLeftOpenClose.commands.commandHomePos, int1 := #HipotTabContactorLeftOpenClose_Inpos[1]."Int"[1], int2 :=, int3 :=, int4 :=, int5 :=, int6 :=, int7 :=, int8 :=, int9 :=, int10 :=, Bypass := #unitStatus.specialFunctions."Spare 35", intOut := "Unit1.Em8.HmiInterface".intCondition.Actuator_53.intOut, Moveing_INT => "Unit1.Em8.ControlNodes".cm.interlock.hipotTabContactorLeft.home)
   END_RUNG
   RUNG wire#powerrail
      I_Contact( "Unit1.Em8.ControlNodes".hipotThickness."step".action1[120] )
      I_Contact( "Unit1.Em8.ControlNodes".hipotThickness."step".action1[362] )
      I_Contact( "Unit1.Em8.ControlNodes".GRnR_hipotThickness."step".action1[362] )
      Not()
      Coil( "Unit1.Em8.ControlNodes".cmHipotTabContactorLeftOpenClose.commands.commandHomePos )
   END_RUNG
   // the same network as SCL:
   #HipotTabContactorLeftOpenClose_Inpos[1]."Int"[1] := NOT #FALSE;
   #instCmHipotTabContactorLeftOpenCloseInterlock[1](Status := #unitStatus,   // "LER_Actuator"
                           HMI := "Unit1.Em8.HmiInterface".cmHipotTabContactorLeftOpenClose.commands.commandHomePos,
                           Process := "Unit1.Em8.ControlNodes".cmHipotTabContactorLeftOpenClose.commands.commandHomePos,
                           int1 := #HipotTabContactorLeftOpenClose_Inpos[1]."Int"[1],
                           Bypass := #unitStatus.specialFunctions."Spare 35",
                           intOut := "Unit1.Em8.HmiInterface".intCondition.Actuator_53.intOut,
                           Moveing_INT => "Unit1.Em8.ControlNodes".cm.interlock.hipotTabContactorLeft.home);
   "Unit1.Em8.ControlNodes".cmHipotTabContactorLeftOpenClose.commands.commandHomePos := NOT (NOT "Unit1.Em8.ControlNodes".hipotThickness."step".action1[120] AND NOT "Unit1.Em8.ControlNodes".hipotThickness."step".action1[362] AND NOT "Unit1.Em8.ControlNodes".GRnR_hipotThickness."step".action1[362]);
END_REGION

REGION Network 88: Hipot Tab Contactor Left Commands
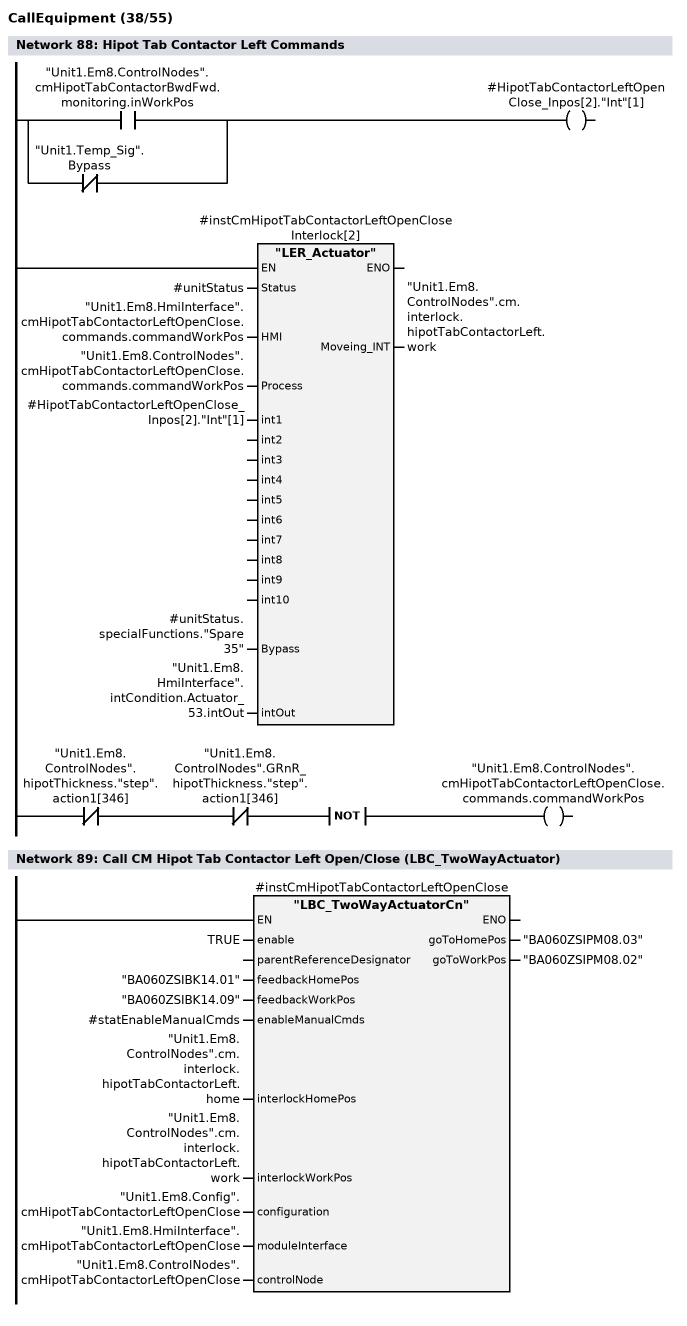
   RUNG wire#powerrail
      Contact( "Unit1.Em8.ControlNodes".cmHipotTabContactorBwdFwd.monitoring.inWorkPos )
      wire#w1
      Coil( #HipotTabContactorLeftOpenClose_Inpos[2]."Int"[1] )
   END_RUNG
   RUNG wire#powerrail
      I_Contact( "Unit1.Temp_Sig".Bypass )
   END_RUNG wire#w1
   RUNG wire#powerrail
      #instCmHipotTabContactorLeftOpenCloseInterlock[2](Status := #unitStatus, HMI := "Unit1.Em8.HmiInterface".cmHipotTabContactorLeftOpenClose.commands.commandWorkPos, Process := "Unit1.Em8.ControlNodes".cmHipotTabContactorLeftOpenClose.commands.commandWorkPos, int1 := #HipotTabContactorLeftOpenClose_Inpos[2]."Int"[1], int2 :=, int3 :=, int4 :=, int5 :=, int6 :=, int7 :=, int8 :=, int9 :=, int10 :=, Bypass := #unitStatus.specialFunctions."Spare 35", intOut := "Unit1.Em8.HmiInterface".intCondition.Actuator_53.intOut, Moveing_INT => "Unit1.Em8.ControlNodes".cm.interlock.hipotTabContactorLeft.work)
   END_RUNG
   RUNG wire#powerrail
      I_Contact( "Unit1.Em8.ControlNodes".hipotThickness."step".action1[346] )
      I_Contact( "Unit1.Em8.ControlNodes".GRnR_hipotThickness."step".action1[346] )
      Not()
      Coil( "Unit1.Em8.ControlNodes".cmHipotTabContactorLeftOpenClose.commands.commandWorkPos )
   END_RUNG
   // the same network as SCL:
   #HipotTabContactorLeftOpenClose_Inpos[2]."Int"[1] := "Unit1.Em8.ControlNodes".cmHipotTabContactorBwdFwd.monitoring.inWorkPos OR NOT "Unit1.Temp_Sig".Bypass;
   #instCmHipotTabContactorLeftOpenCloseInterlock[2](Status := #unitStatus,   // "LER_Actuator"
                           HMI := "Unit1.Em8.HmiInterface".cmHipotTabContactorLeftOpenClose.commands.commandWorkPos,
                           Process := "Unit1.Em8.ControlNodes".cmHipotTabContactorLeftOpenClose.commands.commandWorkPos,
                           int1 := #HipotTabContactorLeftOpenClose_Inpos[2]."Int"[1],
                           Bypass := #unitStatus.specialFunctions."Spare 35",
                           intOut := "Unit1.Em8.HmiInterface".intCondition.Actuator_53.intOut,
                           Moveing_INT => "Unit1.Em8.ControlNodes".cm.interlock.hipotTabContactorLeft.work);
   "Unit1.Em8.ControlNodes".cmHipotTabContactorLeftOpenClose.commands.commandWorkPos := NOT (NOT "Unit1.Em8.ControlNodes".hipotThickness."step".action1[346] AND NOT "Unit1.Em8.ControlNodes".GRnR_hipotThickness."step".action1[346]);
END_REGION

REGION Network 89: Call CM Hipot Tab Contactor Left Open/Close (LBC_TwoWayActuator)
   RUNG wire#powerrail
      #instCmHipotTabContactorLeftOpenClose(enable := TRUE, parentReferenceDesignator :=, feedbackHomePos := "BA060ZSIBK14.01", feedbackWorkPos := "BA060ZSIBK14.09", enableManualCmds := #statEnableManualCmds, interlockHomePos := "Unit1.Em8.ControlNodes".cm.interlock.hipotTabContactorLeft.home, interlockWorkPos := "Unit1.Em8.ControlNodes".cm.interlock.hipotTabContactorLeft.work, configuration := "Unit1.Em8.Config".cmHipotTabContactorLeftOpenClose, moduleInterface := "Unit1.Em8.HmiInterface".cmHipotTabContactorLeftOpenClose, controlNode := "Unit1.Em8.ControlNodes".cmHipotTabContactorLeftOpenClose, goToHomePos => "BA060ZSIPM08.03", goToWorkPos => "BA060ZSIPM08.02")
   END_RUNG
   // the same network as SCL:
   #instCmHipotTabContactorLeftOpenClose(enable := TRUE,   // "LBC_TwoWayActuatorCn"
                           feedbackHomePos := "BA060ZSIBK14.01",
                           feedbackWorkPos := "BA060ZSIBK14.09",
                           enableManualCmds := #statEnableManualCmds,
                           interlockHomePos := "Unit1.Em8.ControlNodes".cm.interlock.hipotTabContactorLeft.home,
                           interlockWorkPos := "Unit1.Em8.ControlNodes".cm.interlock.hipotTabContactorLeft.work,
                           configuration := "Unit1.Em8.Config".cmHipotTabContactorLeftOpenClose,
                           moduleInterface := "Unit1.Em8.HmiInterface".cmHipotTabContactorLeftOpenClose,
                           controlNode := "Unit1.Em8.ControlNodes".cmHipotTabContactorLeftOpenClose,
                           goToHomePos => "BA060ZSIPM08.03",
                           goToWorkPos => "BA060ZSIPM08.02");
END_REGION

REGION Network 91: Hipot Tab Contactor Right Interlock Condition
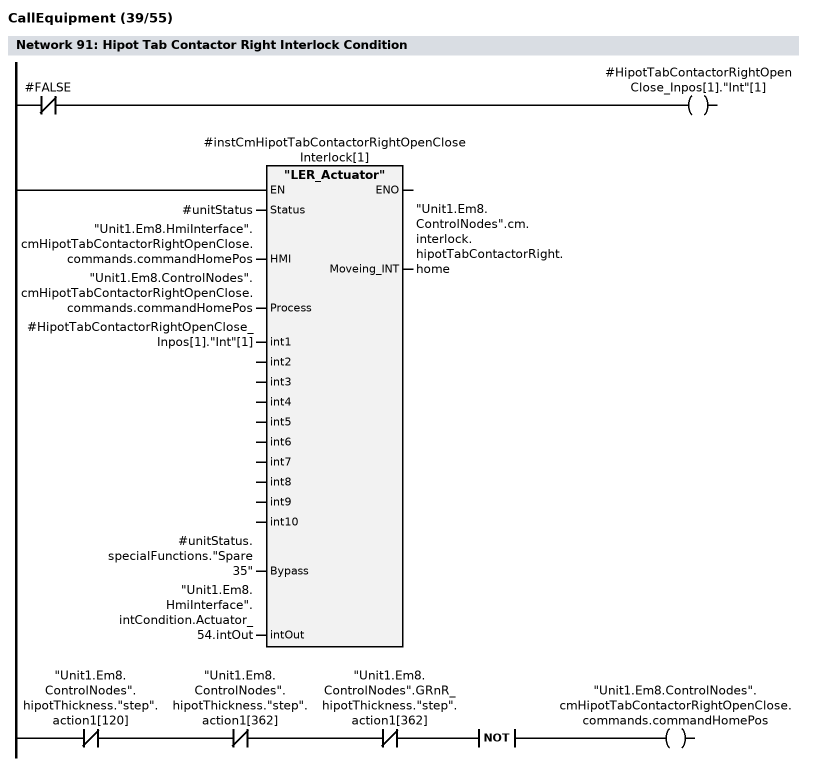
   RUNG wire#powerrail
      I_Contact( #FALSE )
      Coil( #HipotTabContactorRightOpenClose_Inpos[1]."Int"[1] )
   END_RUNG
   RUNG wire#powerrail
      #instCmHipotTabContactorRightOpenCloseInterlock[1](Status := #unitStatus, HMI := "Unit1.Em8.HmiInterface".cmHipotTabContactorRightOpenClose.commands.commandHomePos, Process := "Unit1.Em8.ControlNodes".cmHipotTabContactorRightOpenClose.commands.commandHomePos, int1 := #HipotTabContactorRightOpenClose_Inpos[1]."Int"[1], int2 :=, int3 :=, int4 :=, int5 :=, int6 :=, int7 :=, int8 :=, int9 :=, int10 :=, Bypass := #unitStatus.specialFunctions."Spare 35", intOut := "Unit1.Em8.HmiInterface".intCondition.Actuator_54.intOut, Moveing_INT => "Unit1.Em8.ControlNodes".cm.interlock.hipotTabContactorRight.home)
   END_RUNG
   RUNG wire#powerrail
      I_Contact( "Unit1.Em8.ControlNodes".hipotThickness."step".action1[120] )
      I_Contact( "Unit1.Em8.ControlNodes".hipotThickness."step".action1[362] )
      I_Contact( "Unit1.Em8.ControlNodes".GRnR_hipotThickness."step".action1[362] )
      Not()
      Coil( "Unit1.Em8.ControlNodes".cmHipotTabContactorRightOpenClose.commands.commandHomePos )
   END_RUNG
   // the same network as SCL:
   #HipotTabContactorRightOpenClose_Inpos[1]."Int"[1] := NOT #FALSE;
   #instCmHipotTabContactorRightOpenCloseInterlock[1](Status := #unitStatus,   // "LER_Actuator"
                           HMI := "Unit1.Em8.HmiInterface".cmHipotTabContactorRightOpenClose.commands.commandHomePos,
                           Process := "Unit1.Em8.ControlNodes".cmHipotTabContactorRightOpenClose.commands.commandHomePos,
                           int1 := #HipotTabContactorRightOpenClose_Inpos[1]."Int"[1],
                           Bypass := #unitStatus.specialFunctions."Spare 35",
                           intOut := "Unit1.Em8.HmiInterface".intCondition.Actuator_54.intOut,
                           Moveing_INT => "Unit1.Em8.ControlNodes".cm.interlock.hipotTabContactorRight.home);
   "Unit1.Em8.ControlNodes".cmHipotTabContactorRightOpenClose.commands.commandHomePos := NOT (NOT "Unit1.Em8.ControlNodes".hipotThickness."step".action1[120] AND NOT "Unit1.Em8.ControlNodes".hipotThickness."step".action1[362] AND NOT "Unit1.Em8.ControlNodes".GRnR_hipotThickness."step".action1[362]);
END_REGION

REGION Network 92: Hipot Tab Contactor Right Commands
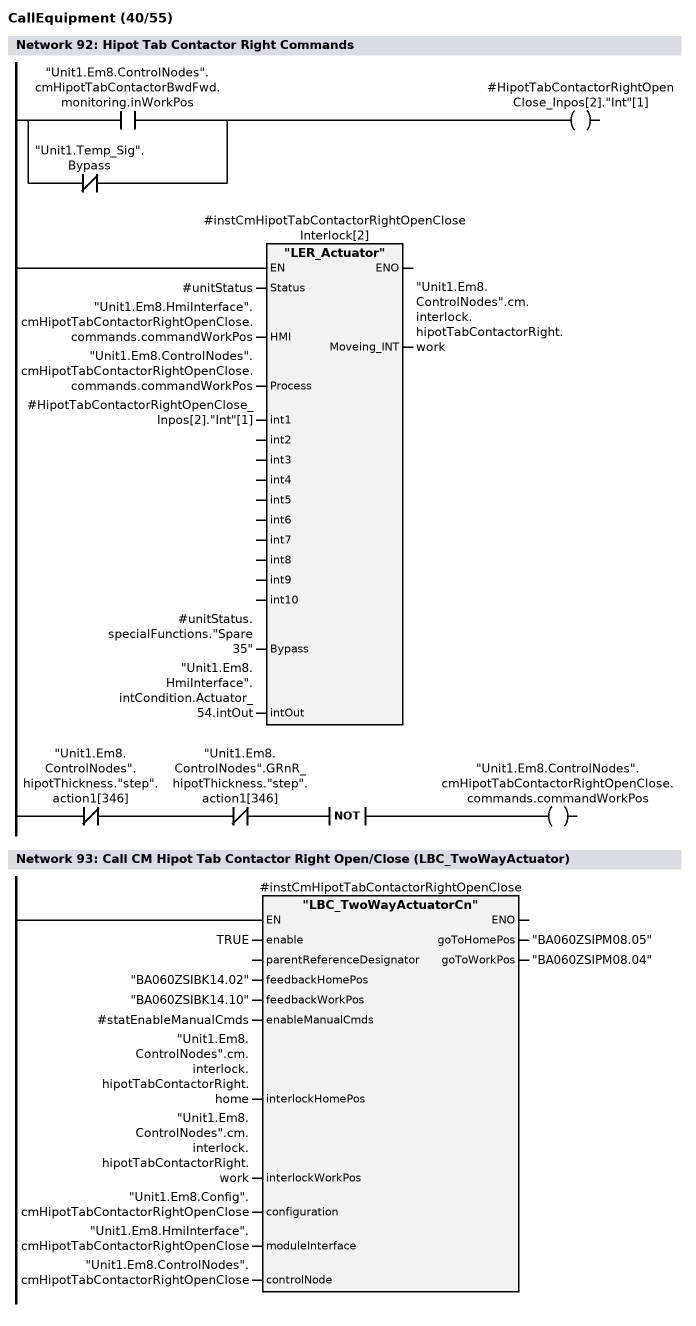
   RUNG wire#powerrail
      Contact( "Unit1.Em8.ControlNodes".cmHipotTabContactorBwdFwd.monitoring.inWorkPos )
      wire#w1
      Coil( #HipotTabContactorRightOpenClose_Inpos[2]."Int"[1] )
   END_RUNG
   RUNG wire#powerrail
      I_Contact( "Unit1.Temp_Sig".Bypass )
   END_RUNG wire#w1
   RUNG wire#powerrail
      #instCmHipotTabContactorRightOpenCloseInterlock[2](Status := #unitStatus, HMI := "Unit1.Em8.HmiInterface".cmHipotTabContactorRightOpenClose.commands.commandWorkPos, Process := "Unit1.Em8.ControlNodes".cmHipotTabContactorRightOpenClose.commands.commandWorkPos, int1 := #HipotTabContactorRightOpenClose_Inpos[2]."Int"[1], int2 :=, int3 :=, int4 :=, int5 :=, int6 :=, int7 :=, int8 :=, int9 :=, int10 :=, Bypass := #unitStatus.specialFunctions."Spare 35", intOut := "Unit1.Em8.HmiInterface".intCondition.Actuator_54.intOut, Moveing_INT => "Unit1.Em8.ControlNodes".cm.interlock.hipotTabContactorRight.work)
   END_RUNG
   RUNG wire#powerrail
      I_Contact( "Unit1.Em8.ControlNodes".hipotThickness."step".action1[346] )
      I_Contact( "Unit1.Em8.ControlNodes".GRnR_hipotThickness."step".action1[346] )
      Not()
      Coil( "Unit1.Em8.ControlNodes".cmHipotTabContactorRightOpenClose.commands.commandWorkPos )
   END_RUNG
   // the same network as SCL:
   #HipotTabContactorRightOpenClose_Inpos[2]."Int"[1] := "Unit1.Em8.ControlNodes".cmHipotTabContactorBwdFwd.monitoring.inWorkPos OR NOT "Unit1.Temp_Sig".Bypass;
   #instCmHipotTabContactorRightOpenCloseInterlock[2](Status := #unitStatus,   // "LER_Actuator"
                           HMI := "Unit1.Em8.HmiInterface".cmHipotTabContactorRightOpenClose.commands.commandWorkPos,
                           Process := "Unit1.Em8.ControlNodes".cmHipotTabContactorRightOpenClose.commands.commandWorkPos,
                           int1 := #HipotTabContactorRightOpenClose_Inpos[2]."Int"[1],
                           Bypass := #unitStatus.specialFunctions."Spare 35",
                           intOut := "Unit1.Em8.HmiInterface".intCondition.Actuator_54.intOut,
                           Moveing_INT => "Unit1.Em8.ControlNodes".cm.interlock.hipotTabContactorRight.work);
   "Unit1.Em8.ControlNodes".cmHipotTabContactorRightOpenClose.commands.commandWorkPos := NOT (NOT "Unit1.Em8.ControlNodes".hipotThickness."step".action1[346] AND NOT "Unit1.Em8.ControlNodes".GRnR_hipotThickness."step".action1[346]);
END_REGION

REGION Network 93: Call CM Hipot Tab Contactor Right Open/Close (LBC_TwoWayActuator)
   RUNG wire#powerrail
      #instCmHipotTabContactorRightOpenClose(enable := TRUE, parentReferenceDesignator :=, feedbackHomePos := "BA060ZSIBK14.02", feedbackWorkPos := "BA060ZSIBK14.10", enableManualCmds := #statEnableManualCmds, interlockHomePos := "Unit1.Em8.ControlNodes".cm.interlock.hipotTabContactorRight.home, interlockWorkPos := "Unit1.Em8.ControlNodes".cm.interlock.hipotTabContactorRight.work, configuration := "Unit1.Em8.Config".cmHipotTabContactorRightOpenClose, moduleInterface := "Unit1.Em8.HmiInterface".cmHipotTabContactorRightOpenClose, controlNode := "Unit1.Em8.ControlNodes".cmHipotTabContactorRightOpenClose, goToHomePos => "BA060ZSIPM08.05", goToWorkPos => "BA060ZSIPM08.04")
   END_RUNG
   // the same network as SCL:
   #instCmHipotTabContactorRightOpenClose(enable := TRUE,   // "LBC_TwoWayActuatorCn"
                           feedbackHomePos := "BA060ZSIBK14.02",
                           feedbackWorkPos := "BA060ZSIBK14.10",
                           enableManualCmds := #statEnableManualCmds,
                           interlockHomePos := "Unit1.Em8.ControlNodes".cm.interlock.hipotTabContactorRight.home,
                           interlockWorkPos := "Unit1.Em8.ControlNodes".cm.interlock.hipotTabContactorRight.work,
                           configuration := "Unit1.Em8.Config".cmHipotTabContactorRightOpenClose,
                           moduleInterface := "Unit1.Em8.HmiInterface".cmHipotTabContactorRightOpenClose,
                           controlNode := "Unit1.Em8.ControlNodes".cmHipotTabContactorRightOpenClose,
                           goToHomePos => "BA060ZSIPM08.05",
                           goToWorkPos => "BA060ZSIPM08.04");
END_REGION

REGION Network 95: Hipot & Thickness Stage Lift All Interlock Condition
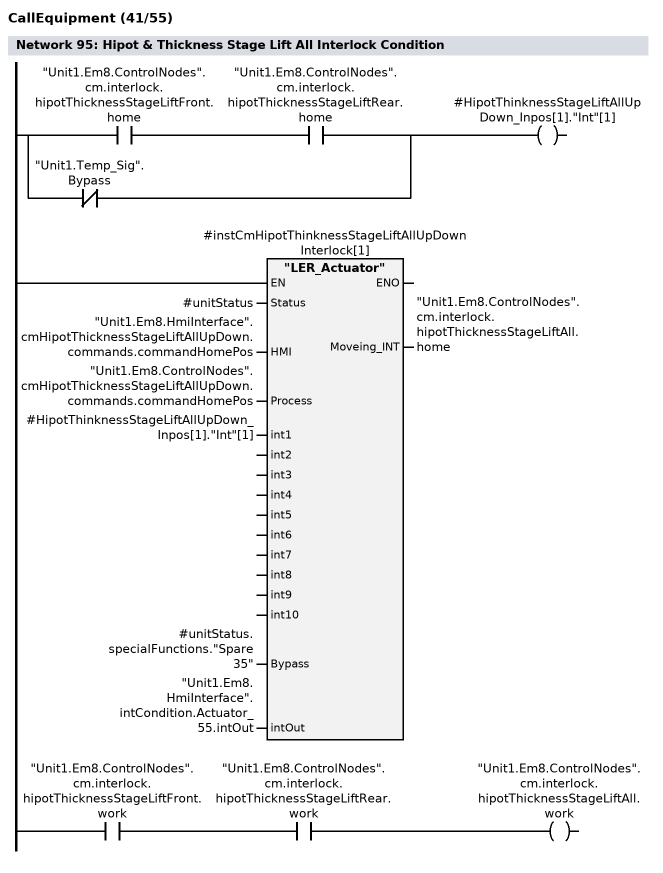
   RUNG wire#powerrail
      Contact( "Unit1.Em8.ControlNodes".cm.interlock.hipotThicknessStageLiftFront.home )
      Contact( "Unit1.Em8.ControlNodes".cm.interlock.hipotThicknessStageLiftRear.home )
      wire#w1
      Coil( #HipotThinknessStageLiftAllUpDown_Inpos[1]."Int"[1] )
   END_RUNG
   RUNG wire#powerrail
      I_Contact( "Unit1.Temp_Sig".Bypass )
   END_RUNG wire#w1
   RUNG wire#powerrail
      #instCmHipotThinknessStageLiftAllUpDownInterlock[1](Status := #unitStatus, HMI := "Unit1.Em8.HmiInterface".cmHipotThicknessStageLiftAllUpDown.commands.commandHomePos, Process := "Unit1.Em8.ControlNodes".cmHipotThicknessStageLiftAllUpDown.commands.commandHomePos, int1 := #HipotThinknessStageLiftAllUpDown_Inpos[1]."Int"[1], int2 :=, int3 :=, int4 :=, int5 :=, int6 :=, int7 :=, int8 :=, int9 :=, int10 :=, Bypass := #unitStatus.specialFunctions."Spare 35", intOut := "Unit1.Em8.HmiInterface".intCondition.Actuator_55.intOut, Moveing_INT => "Unit1.Em8.ControlNodes".cm.interlock.hipotThicknessStageLiftAll.home)
   END_RUNG
   RUNG wire#powerrail
      Contact( "Unit1.Em8.ControlNodes".cm.interlock.hipotThicknessStageLiftFront.work )
      Contact( "Unit1.Em8.ControlNodes".cm.interlock.hipotThicknessStageLiftRear.work )
      Coil( "Unit1.Em8.ControlNodes".cm.interlock.hipotThicknessStageLiftAll.work )
   END_RUNG
   // the same network as SCL:
   #HipotThinknessStageLiftAllUpDown_Inpos[1]."Int"[1] := ("Unit1.Em8.ControlNodes".cm.interlock.hipotThicknessStageLiftFront.home AND "Unit1.Em8.ControlNodes".cm.interlock.hipotThicknessStageLiftRear.home) OR NOT "Unit1.Temp_Sig".Bypass;
   #instCmHipotThinknessStageLiftAllUpDownInterlock[1](Status := #unitStatus,   // "LER_Actuator"
                           HMI := "Unit1.Em8.HmiInterface".cmHipotThicknessStageLiftAllUpDown.commands.commandHomePos,
                           Process := "Unit1.Em8.ControlNodes".cmHipotThicknessStageLiftAllUpDown.commands.commandHomePos,
                           int1 := #HipotThinknessStageLiftAllUpDown_Inpos[1]."Int"[1],
                           Bypass := #unitStatus.specialFunctions."Spare 35",
                           intOut := "Unit1.Em8.HmiInterface".intCondition.Actuator_55.intOut,
                           Moveing_INT => "Unit1.Em8.ControlNodes".cm.interlock.hipotThicknessStageLiftAll.home);
   "Unit1.Em8.ControlNodes".cm.interlock.hipotThicknessStageLiftAll.work := "Unit1.Em8.ControlNodes".cm.interlock.hipotThicknessStageLiftFront.work AND "Unit1.Em8.ControlNodes".cm.interlock.hipotThicknessStageLiftRear.work;
END_REGION

REGION Network 96: Hipot & Thickness Stage Lift All Interlock Condition
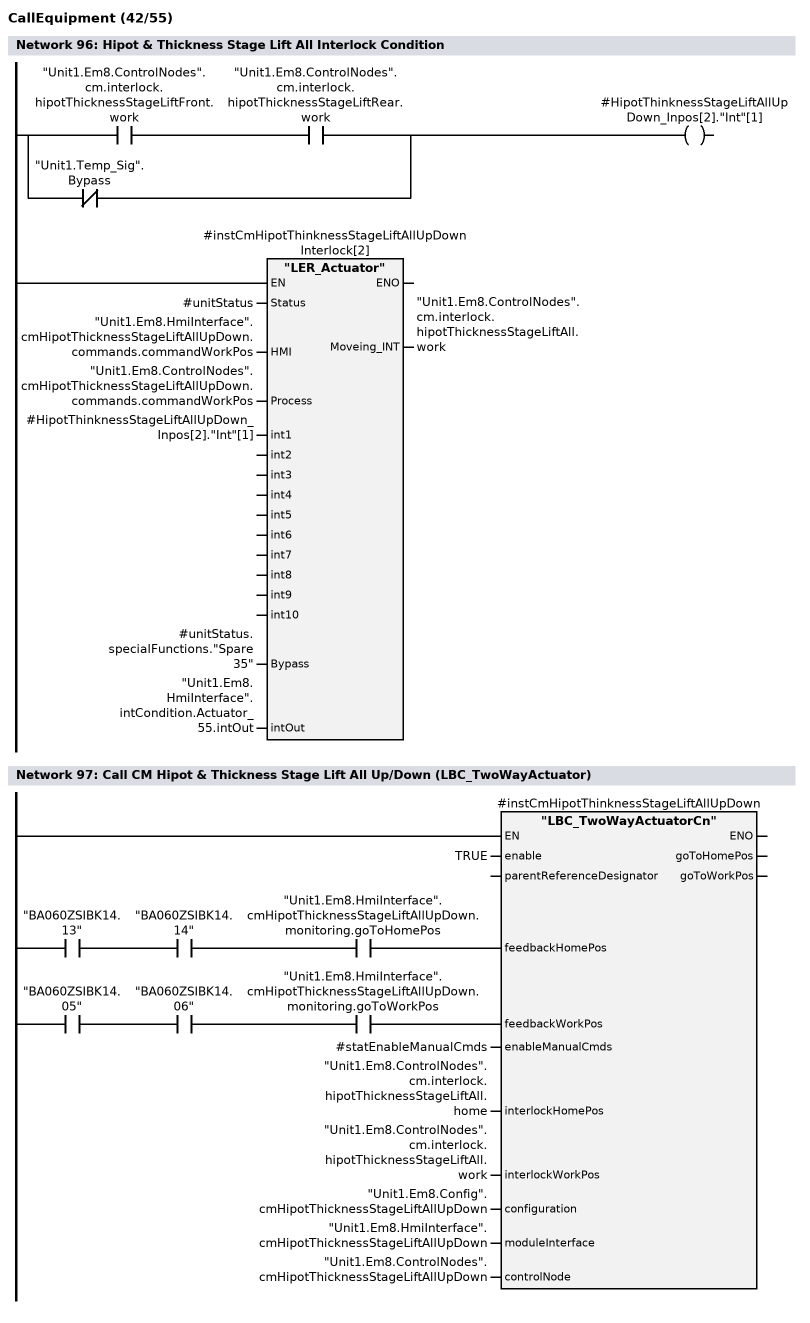
   RUNG wire#powerrail
      Contact( "Unit1.Em8.ControlNodes".cm.interlock.hipotThicknessStageLiftFront.work )
      Contact( "Unit1.Em8.ControlNodes".cm.interlock.hipotThicknessStageLiftRear.work )
      wire#w1
      Coil( #HipotThinknessStageLiftAllUpDown_Inpos[2]."Int"[1] )
   END_RUNG
   RUNG wire#powerrail
      I_Contact( "Unit1.Temp_Sig".Bypass )
   END_RUNG wire#w1
   RUNG wire#powerrail
      #instCmHipotThinknessStageLiftAllUpDownInterlock[2](Status := #unitStatus, HMI := "Unit1.Em8.HmiInterface".cmHipotThicknessStageLiftAllUpDown.commands.commandWorkPos, Process := "Unit1.Em8.ControlNodes".cmHipotThicknessStageLiftAllUpDown.commands.commandWorkPos, int1 := #HipotThinknessStageLiftAllUpDown_Inpos[2]."Int"[1], int2 :=, int3 :=, int4 :=, int5 :=, int6 :=, int7 :=, int8 :=, int9 :=, int10 :=, Bypass := #unitStatus.specialFunctions."Spare 35", intOut := "Unit1.Em8.HmiInterface".intCondition.Actuator_55.intOut, Moveing_INT => "Unit1.Em8.ControlNodes".cm.interlock.hipotThicknessStageLiftAll.work)
   END_RUNG
   // the same network as SCL:
   #HipotThinknessStageLiftAllUpDown_Inpos[2]."Int"[1] := ("Unit1.Em8.ControlNodes".cm.interlock.hipotThicknessStageLiftFront.work AND "Unit1.Em8.ControlNodes".cm.interlock.hipotThicknessStageLiftRear.work) OR NOT "Unit1.Temp_Sig".Bypass;
   #instCmHipotThinknessStageLiftAllUpDownInterlock[2](Status := #unitStatus,   // "LER_Actuator"
                           HMI := "Unit1.Em8.HmiInterface".cmHipotThicknessStageLiftAllUpDown.commands.commandWorkPos,
                           Process := "Unit1.Em8.ControlNodes".cmHipotThicknessStageLiftAllUpDown.commands.commandWorkPos,
                           int1 := #HipotThinknessStageLiftAllUpDown_Inpos[2]."Int"[1],
                           Bypass := #unitStatus.specialFunctions."Spare 35",
                           intOut := "Unit1.Em8.HmiInterface".intCondition.Actuator_55.intOut,
                           Moveing_INT => "Unit1.Em8.ControlNodes".cm.interlock.hipotThicknessStageLiftAll.work);
END_REGION

REGION Network 97: Call CM Hipot & Thickness Stage Lift All Up/Down (LBC_TwoWayActuator)
   RUNG wire#powerrail
      #instCmHipotThinknessStageLiftAllUpDown(feedbackHomePos := wire#w1, feedbackWorkPos := wire#w2, enable := TRUE, parentReferenceDesignator :=, enableManualCmds := #statEnableManualCmds, interlockHomePos := "Unit1.Em8.ControlNodes".cm.interlock.hipotThicknessStageLiftAll.home, interlockWorkPos := "Unit1.Em8.ControlNodes".cm.interlock.hipotThicknessStageLiftAll.work, configuration := "Unit1.Em8.Config".cmHipotThicknessStageLiftAllUpDown, moduleInterface := "Unit1.Em8.HmiInterface".cmHipotThicknessStageLiftAllUpDown, controlNode := "Unit1.Em8.ControlNodes".cmHipotThicknessStageLiftAllUpDown, goToHomePos =>, goToWorkPos =>)
   END_RUNG
   RUNG wire#powerrail
      Contact( "BA060ZSIBK14.13" )
      Contact( "BA060ZSIBK14.14" )
      Contact( "Unit1.Em8.HmiInterface".cmHipotThicknessStageLiftAllUpDown.monitoring.goToHomePos )
   END_RUNG wire#w1
   RUNG wire#powerrail
      Contact( "BA060ZSIBK14.05" )
      Contact( "BA060ZSIBK14.06" )
      Contact( "Unit1.Em8.HmiInterface".cmHipotThicknessStageLiftAllUpDown.monitoring.goToWorkPos )
   END_RUNG wire#w2
   // the same network as SCL:
   #instCmHipotThinknessStageLiftAllUpDown(enable := TRUE,   // "LBC_TwoWayActuatorCn"
                           feedbackHomePos := "BA060ZSIBK14.13" AND "BA060ZSIBK14.14" AND "Unit1.Em8.HmiInterface".cmHipotThicknessStageLiftAllUpDown.monitoring.goToHomePos,
                           feedbackWorkPos := "BA060ZSIBK14.05" AND "BA060ZSIBK14.06" AND "Unit1.Em8.HmiInterface".cmHipotThicknessStageLiftAllUpDown.monitoring.goToWorkPos,
                           enableManualCmds := #statEnableManualCmds,
                           interlockHomePos := "Unit1.Em8.ControlNodes".cm.interlock.hipotThicknessStageLiftAll.home,
                           interlockWorkPos := "Unit1.Em8.ControlNodes".cm.interlock.hipotThicknessStageLiftAll.work,
                           configuration := "Unit1.Em8.Config".cmHipotThicknessStageLiftAllUpDown,
                           moduleInterface := "Unit1.Em8.HmiInterface".cmHipotThicknessStageLiftAllUpDown,
                           controlNode := "Unit1.Em8.ControlNodes".cmHipotThicknessStageLiftAllUpDown);
END_REGION

REGION Network 99: ******************** Control Modules (Accessories) ********************
END_REGION

REGION Network 100: Thickness Control Commands
